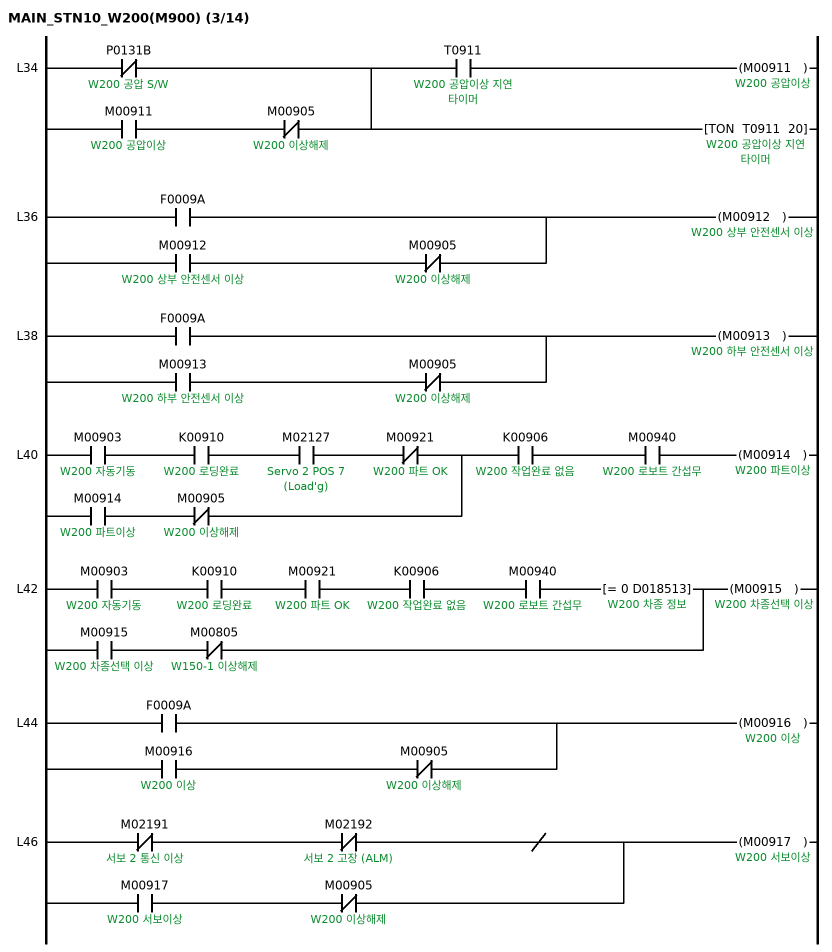
[picture p168: MAIN_STN10_W200(M900) rungs L34-L46]
; L34
LOAD NOT  P0131B	// W200 공압 S/W
LOAD      M00911	// W200 공압이상
AND NOT   M00905	// W200 이상해제
OR LOAD
MPUSH
AND       T0911	// W200 공압이상 지연 타이머
OUT       M00911	// W200 공압이상
MPOP
TON       T0911 20	// W200 공압이상 지연 타이머
; L36
LOAD      F0009A
LOAD      M00912	// W200 상부 안전센서 이상
AND NOT   M00905	// W200 이상해제
OR LOAD
OUT       M00912	// W200 상부 안전센서 이상
; L38
LOAD      F0009A
LOAD      M00913	// W200 하부 안전센서 이상
AND NOT   M00905	// W200 이상해제
OR LOAD
OUT       M00913	// W200 하부 안전센서 이상
; L40
LOAD      M00903	// W200 자동기동
AND       K00910	// W200 로딩완료
AND       M02127	// Servo 2 POS 7 (Load'g)
AND NOT   M00921	// W200 파트 OK
LOAD      M00914	// W200 파트이상
AND NOT   M00905	// W200 이상해제
OR LOAD
AND       K00906	// W200 작업완료 없음
AND       M00940	// W200 로보트 간섭무
OUT       M00914	// W200 파트이상
; L42
LOAD      M00903	// W200 자동기동
AND       K00910	// W200 로딩완료
AND       M00921	// W200 파트 OK
AND       K00906	// W200 작업완료 없음
AND       M00940	// W200 로보트 간섭무
AND=      0 D018513	// W200 차종 정보
LOAD      M00915	// W200 차종선택 이상
AND NOT   M00805	// W150-1 이상해제
OR LOAD
OUT       M00915	// W200 차종선택 이상
; L44
LOAD      F0009A
LOAD      M00916	// W200 이상
AND NOT   M00905	// W200 이상해제
OR LOAD
OUT       M00916	// W200 이상
; L46
LOAD NOT  M02191	// 서보 2 통신 이상
AND NOT   M02192	// 서보 2 고장 (ALM)
NOT
LOAD      M00917	// W200 서보이상
AND NOT   M00905	// W200 이상해제
OR LOAD
OUT       M00917	// W200 서보이상

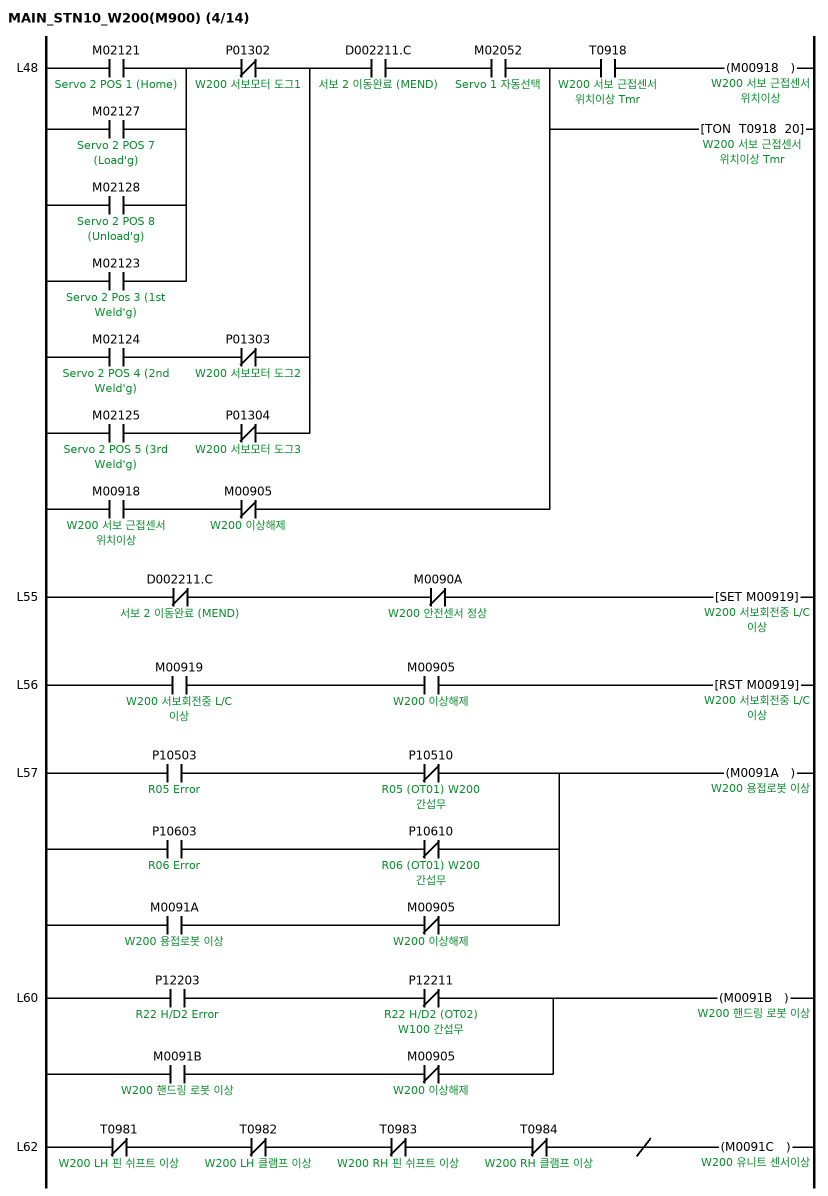
; L48
LOAD      M02121	// Servo 2 POS 1 (Home)
OR        M02127	// Servo 2 POS 7 (Load'g)
OR        M02128	// Servo 2 POS 8 (Unload'g)
OR        M02123	// Servo 2 Pos 3 (1st Weld'g)
AND NOT   P01302	// W200 서보모터 도그1
LOAD      M02124	// Servo 2 POS 4 (2nd Weld'g)
AND NOT   P01303	// W200 서보모터 도그2
OR LOAD
LOAD      M02125	// Servo 2 POS 5 (3rd Weld'g)
AND NOT   P01304	// W200 서보모터 도그3
OR LOAD
AND       D002211.C	// 서보 2 이동완료 (MEND)
AND       M02052	// Servo 1 자동선택
LOAD      M00918	// W200 서보 근접센서 위치이상
AND NOT   M00905	// W200 이상해제
OR LOAD
MPUSH
AND       T0918	// W200 서보 근접센서 위치이상 Tmr
OUT       M00918	// W200 서보 근접센서 위치이상
MPOP
TON       T0918 20	// W200 서보 근접센서 위치이상 Tmr
; L55
LOAD NOT  D002211.C	// 서보 2 이동완료 (MEND)
AND NOT   M0090A	// W200 안전센서 정상
SET       M00919	// W200 서보회전중 L/C 이상
; L56
LOAD      M00919	// W200 서보회전중 L/C 이상
AND       M00905	// W200 이상해제
RST       M00919	// W200 서보회전중 L/C 이상
; L57
LOAD      P10503	// R05 Error
AND NOT   P10510	// R05 (OT01) W200 간섭무
LOAD      P10603	// R06 Error
AND NOT   P10610	// R06 (OT01) W200 간섭무
OR LOAD
LOAD      M0091A	// W200 용접로봇 이상
AND NOT   M00905	// W200 이상해제
OR LOAD
OUT       M0091A	// W200 용접로봇 이상
; L60
LOAD      P12203	// R22 H/D2 Error
AND NOT   P12211	// R22 H/D2 (OT02) W100 간섭무
LOAD      M0091B	// W200 핸드링 로봇 이상
AND NOT   M00905	// W200 이상해제
OR LOAD
OUT       M0091B	// W200 핸드링 로봇 이상
; L62
LOAD NOT  T0981	// W200 LH 핀 쉬프트 이상
AND NOT   T0982	// W200 LH 클램프 이상
AND NOT   T0983	// W200 RH 핀 쉬프트 이상
AND NOT   T0984	// W200 RH 클램프 이상
NOT
OUT       M0091C	// W200 유니트 센서이상

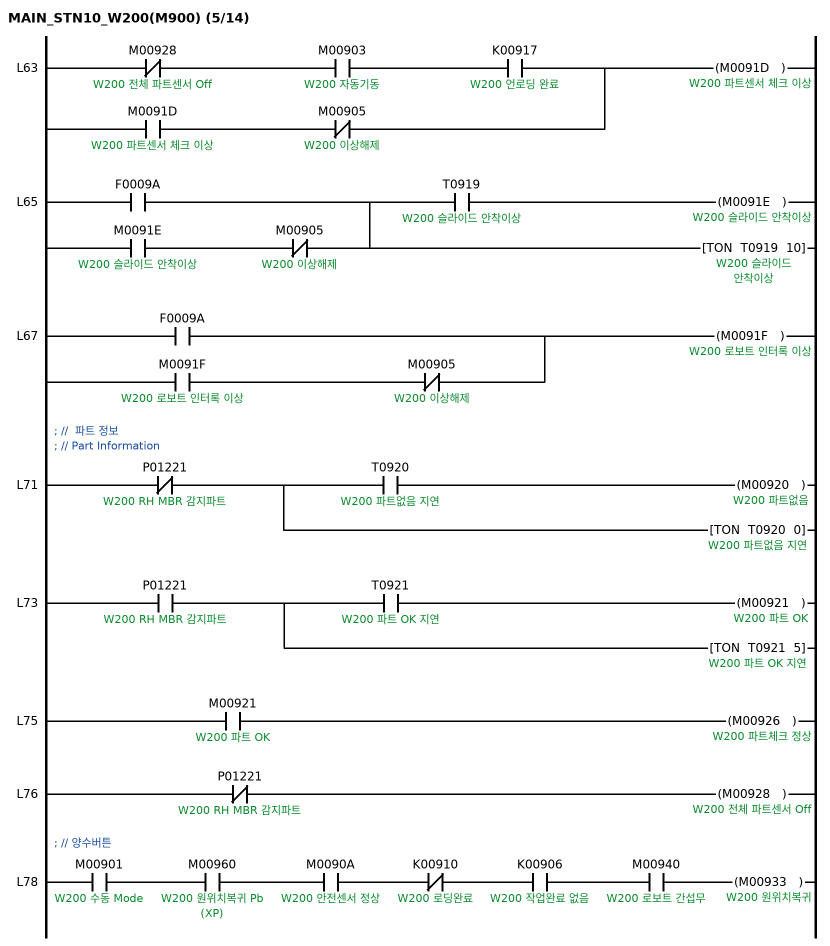
; L63
LOAD NOT  M00928	// W200 전체 파트센서 Off
AND       M00903	// W200 자동기동
AND       K00917	// W200 언로딩 완료
LOAD      M0091D	// W200 파트센서 체크 이상
AND NOT   M00905	// W200 이상해제
OR LOAD
OUT       M0091D	// W200 파트센서 체크 이상
; L65
LOAD      F0009A
LOAD      M0091E	// W200 슬라이드 안착이상
AND NOT   M00905	// W200 이상해제
OR LOAD
MPUSH
AND       T0919	// W200 슬라이드 안착이상
OUT       M0091E	// W200 슬라이드 안착이상
MPOP
TON       T0919 10	// W200 슬라이드 안착이상
; L67
LOAD      F0009A
LOAD      M0091F	// W200 로보트 인터록 이상
AND NOT   M00905	// W200 이상해제
OR LOAD
OUT       M0091F	// W200 로보트 인터록 이상
//   //  파트 정보
//   // Part Information
; L71
LOAD NOT  P01221	// W200 RH MBR 감지파트
MPUSH
AND       T0920	// W200 파트없음 지연
OUT       M00920	// W200 파트없음
MPOP
TON       T0920 0	// W200 파트없음 지연
; L73
LOAD      P01221	// W200 RH MBR 감지파트
MPUSH
AND       T0921	// W200 파트 OK 지연
OUT       M00921	// W200 파트 OK
MPOP
TON       T0921 5	// W200 파트 OK 지연
; L75
LOAD      M00921	// W200 파트 OK
OUT       M00926	// W200 파트체크 정상
; L76
LOAD NOT  P01221	// W200 RH MBR 감지파트
OUT       M00928	// W200 전체 파트센서 Off
//   // 양수버튼
; L78
LOAD      M00901	// W200 수동 Mode
AND       M00960	// W200 원위치복귀 Pb (XP)
AND       M0090A	// W200 안전센서 정상
AND NOT   K00910	// W200 로딩완료
AND       K00906	// W200 작업완료 없음
AND       M00940	// W200 로보트 간섭무
OUT       M00933	// W200 원위치복귀

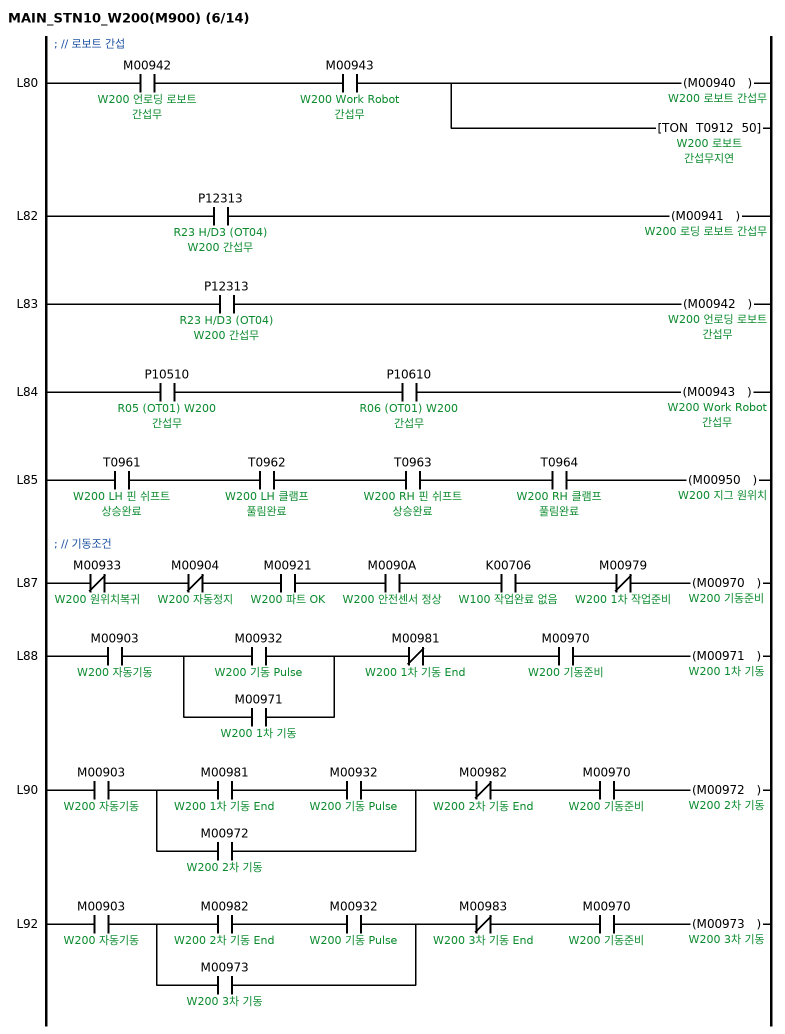
//   // 로보트 간섭
; L80
LOAD      M00942	// W200 언로딩 로보트 간섭무
AND       M00943	// W200 Work Robot 간섭무
OUT       M00940	// W200 로보트 간섭무
TON       T0912 50	// W200 로보트 간섭무지연
; L82
LOAD      P12313	// R23 H/D3 (OT04) W200 간섭무
OUT       M00941	// W200 로딩 로보트 간섭무
; L83
LOAD      P12313	// R23 H/D3 (OT04) W200 간섭무
OUT       M00942	// W200 언로딩 로보트 간섭무
; L84
LOAD      P10510	// R05 (OT01) W200 간섭무
AND       P10610	// R06 (OT01) W200 간섭무
OUT       M00943	// W200 Work Robot 간섭무
; L85
LOAD      T0961	// W200 LH 핀 쉬프트 상승완료
AND       T0962	// W200 LH 클램프 풀림완료
AND       T0963	// W200 RH 핀 쉬프트 상승완료
AND       T0964	// W200 RH 클램프 풀림완료
OUT       M00950	// W200 지그 원위치
//   // 기동조건
; L87
LOAD NOT  M00933	// W200 원위치복귀
AND NOT   M00904	// W200 자동정지
AND       M00921	// W200 파트 OK
AND       M0090A	// W200 안전센서 정상
AND       K00706	// W100 작업완료 없음
AND NOT   M00979	// W200 1차 작업준비
OUT       M00970	// W200 기동준비
; L88
LOAD      M00903	// W200 자동기동
LOAD      M00932	// W200 기동 Pulse
OR        M00971	// W200 1차 기동
AND LOAD
AND NOT   M00981	// W200 1차 기동 End
AND       M00970	// W200 기동준비
OUT       M00971	// W200 1차 기동
; L90
LOAD      M00903	// W200 자동기동
LOAD      M00981	// W200 1차 기동 End
AND       M00932	// W200 기동 Pulse
OR        M00972	// W200 2차 기동
AND LOAD
AND NOT   M00982	// W200 2차 기동 End
AND       M00970	// W200 기동준비
OUT       M00972	// W200 2차 기동
; L92
LOAD      M00903	// W200 자동기동
LOAD      M00982	// W200 2차 기동 End
AND       M00932	// W200 기동 Pulse
OR        M00973	// W200 3차 기동
AND LOAD
AND NOT   M00983	// W200 3차 기동 End
AND       M00970	// W200 기동준비
OUT       M00973	// W200 3차 기동

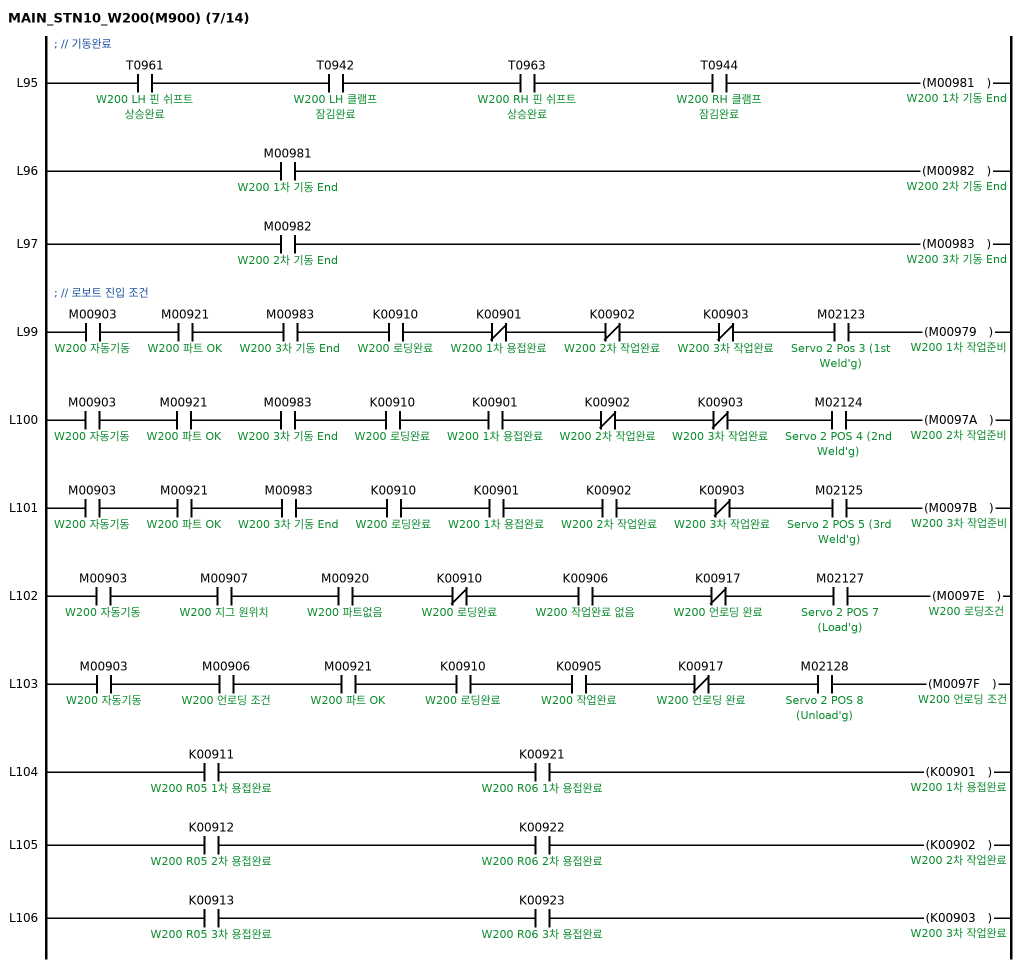
//   // 기동완료
; L95
LOAD      T0961	// W200 LH 핀 쉬프트 상승완료
AND       T0942	// W200 LH 클램프 잠김완료
AND       T0963	// W200 RH 핀 쉬프트 상승완료
AND       T0944	// W200 RH 클램프 잠김완료
OUT       M00981	// W200 1차 기동 End
; L96
LOAD      M00981	// W200 1차 기동 End
OUT       M00982	// W200 2차 기동 End
; L97
LOAD      M00982	// W200 2차 기동 End
OUT       M00983	// W200 3차 기동 End
//   // 로보트 진입 조건
; L99
LOAD      M00903	// W200 자동기동
AND       M00921	// W200 파트 OK
AND       M00983	// W200 3차 기동 End
AND       K00910	// W200 로딩완료
AND NOT   K00901	// W200 1차 용접완료
AND NOT   K00902	// W200 2차 작업완료
AND NOT   K00903	// W200 3차 작업완료
AND       M02123	// Servo 2 Pos 3 (1st Weld'g)
OUT       M00979	// W200 1차 작업준비
; L100
LOAD      M00903	// W200 자동기동
AND       M00921	// W200 파트 OK
AND       M00983	// W200 3차 기동 End
AND       K00910	// W200 로딩완료
AND       K00901	// W200 1차 용접완료
AND NOT   K00902	// W200 2차 작업완료
AND NOT   K00903	// W200 3차 작업완료
AND       M02124	// Servo 2 POS 4 (2nd Weld'g)
OUT       M0097A	// W200 2차 작업준비
; L101
LOAD      M00903	// W200 자동기동
AND       M00921	// W200 파트 OK
AND       M00983	// W200 3차 기동 End
AND       K00910	// W200 로딩완료
AND       K00901	// W200 1차 용접완료
AND       K00902	// W200 2차 작업완료
AND NOT   K00903	// W200 3차 작업완료
AND       M02125	// Servo 2 POS 5 (3rd Weld'g)
OUT       M0097B	// W200 3차 작업준비
; L102
LOAD      M00903	// W200 자동기동
AND       M00907	// W200 지그 원위치
AND       M00920	// W200 파트없음
AND NOT   K00910	// W200 로딩완료
AND       K00906	// W200 작업완료 없음
AND NOT   K00917	// W200 언로딩 완료
AND       M02127	// Servo 2 POS 7 (Load'g)
OUT       M0097E	// W200 로딩조건
; L103
LOAD      M00903	// W200 자동기동
AND       M00906	// W200 언로딩 조건
AND       M00921	// W200 파트 OK
AND       K00910	// W200 로딩완료
AND       K00905	// W200 작업완료
AND NOT   K00917	// W200 언로딩 완료
AND       M02128	// Servo 2 POS 8 (Unload'g)
OUT       M0097F	// W200 언로딩 조건
; L104
LOAD      K00911	// W200 R05 1차 용접완료
AND       K00921	// W200 R06 1차 용접완료
OUT       K00901	// W200 1차 용접완료
; L105
LOAD      K00912	// W200 R05 2차 용접완료
AND       K00922	// W200 R06 2차 용접완료
OUT       K00902	// W200 2차 작업완료
; L106
LOAD      K00913	// W200 R05 3차 용접완료
AND       K00923	// W200 R06 3차 용접완료
OUT       K00903	// W200 3차 작업완료

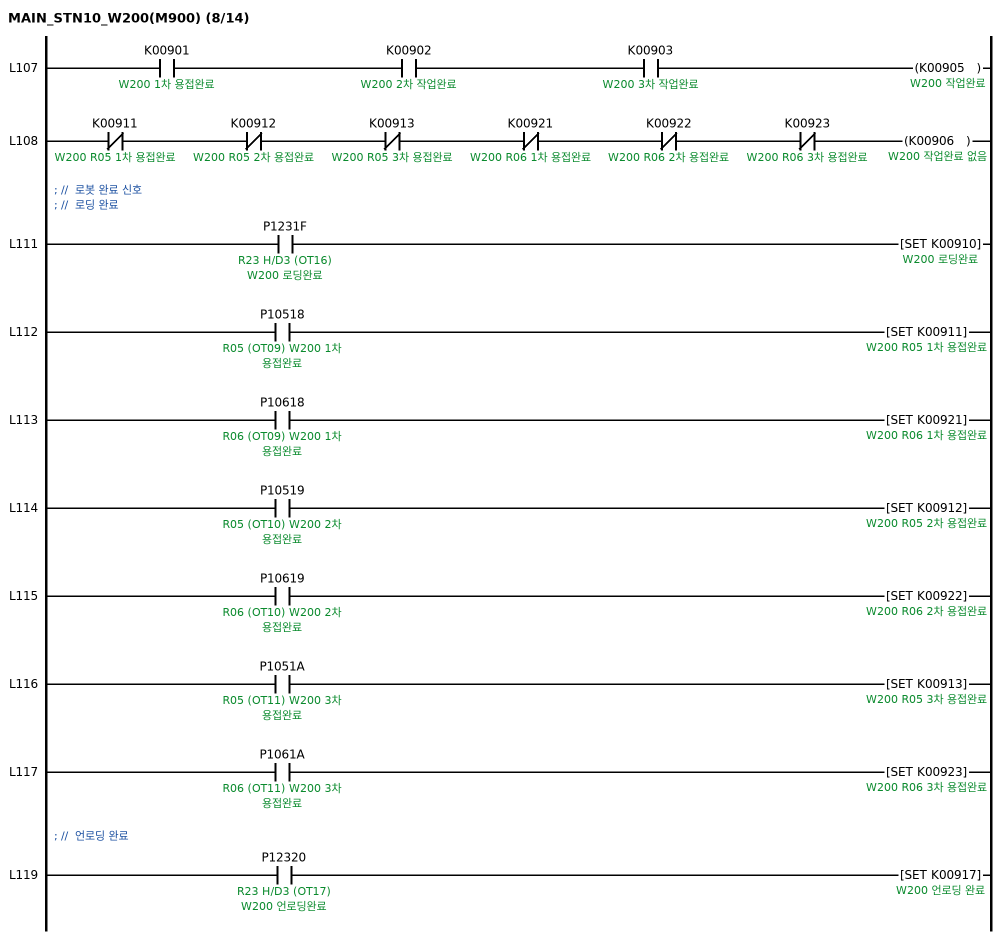
; L107
LOAD      K00901	// W200 1차 용접완료
AND       K00902	// W200 2차 작업완료
AND       K00903	// W200 3차 작업완료
OUT       K00905	// W200 작업완료
; L108
LOAD NOT  K00911	// W200 R05 1차 용접완료
AND NOT   K00912	// W200 R05 2차 용접완료
AND NOT   K00913	// W200 R05 3차 용접완료
AND NOT   K00921	// W200 R06 1차 용접완료
AND NOT   K00922	// W200 R06 2차 용접완료
AND NOT   K00923	// W200 R06 3차 용접완료
OUT       K00906	// W200 작업완료 없음
//   //  로봇 완료 신호
//   //  로딩 완료
; L111
LOAD      P1231F	// R23 H/D3 (OT16) W200 로딩완료
SET       K00910	// W200 로딩완료
; L112
LOAD      P10518	// R05 (OT09) W200 1차 용접완료
SET       K00911	// W200 R05 1차 용접완료
; L113
LOAD      P10618	// R06 (OT09) W200 1차 용접완료
SET       K00921	// W200 R06 1차 용접완료
; L114
LOAD      P10519	// R05 (OT10) W200 2차 용접완료
SET       K00912	// W200 R05 2차 용접완료
; L115
LOAD      P10619	// R06 (OT10) W200 2차 용접완료
SET       K00922	// W200 R06 2차 용접완료
; L116
LOAD      P1051A	// R05 (OT11) W200 3차 용접완료
SET       K00913	// W200 R05 3차 용접완료
; L117
LOAD      P1061A	// R06 (OT11) W200 3차 용접완료
SET       K00923	// W200 R06 3차 용접완료
//   //  언로딩 완료
; L119
LOAD      P12320	// R23 H/D3 (OT17) W200 언로딩완료
SET       K00917	// W200 언로딩 완료

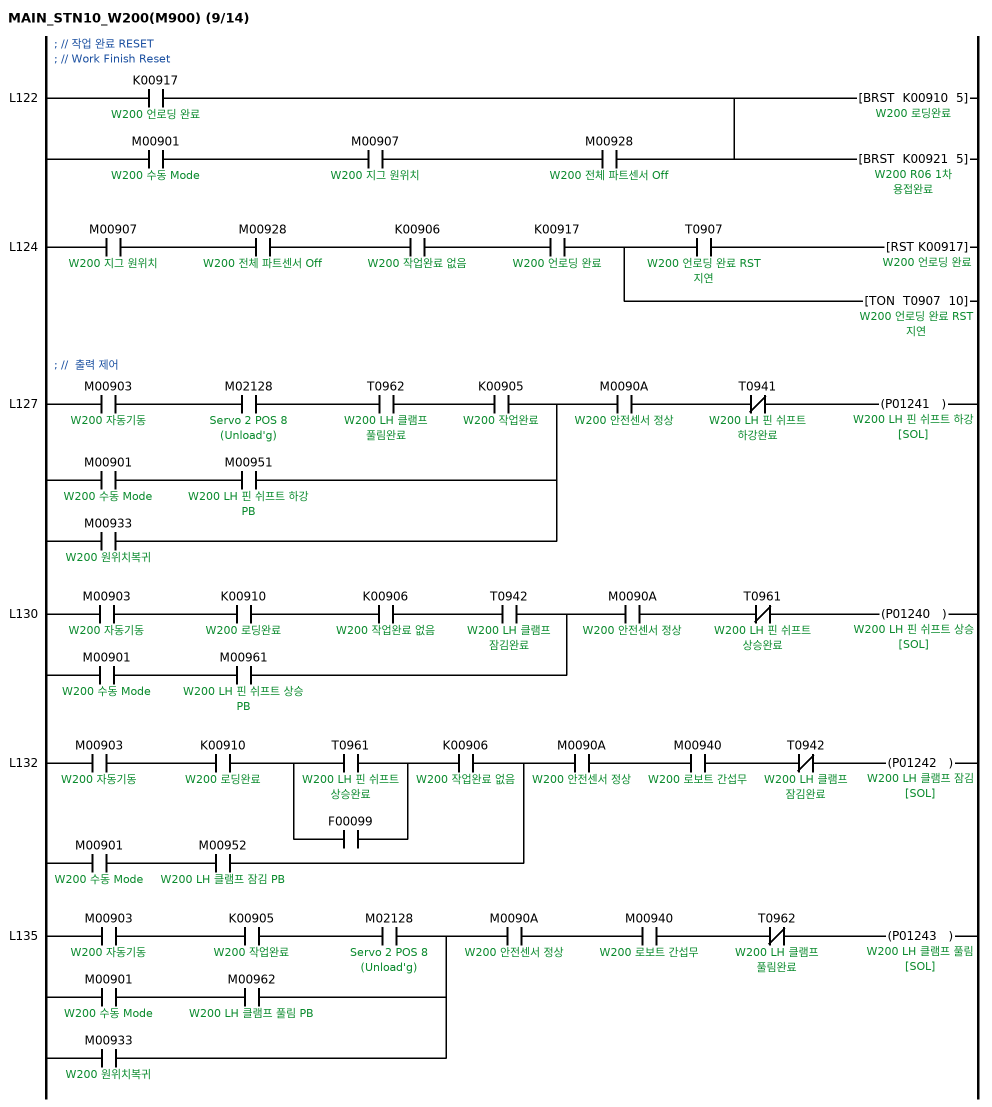
//     // 작업 완료 RESET
//   // Work Finish Reset
; L122
LOAD      K00917	// W200 언로딩 완료
LOAD      M00901	// W200 수동 Mode
AND       M00907	// W200 지그 원위치
AND       M00928	// W200 전체 파트센서 Off
OR LOAD
BRST      K00910 5	// W200 로딩완료
BRST      K00921 5	// W200 R06 1차 용접완료
; L124
LOAD      M00907	// W200 지그 원위치
AND       M00928	// W200 전체 파트센서 Off
AND       K00906	// W200 작업완료 없음
AND       K00917	// W200 언로딩 완료
MPUSH
AND       T0907	// W200 언로딩 완료 RST 지연
RST       K00917	// W200 언로딩 완료
MPOP
TON       T0907 10	// W200 언로딩 완료 RST 지연
//     //  출력 제어
; L127
LOAD      M00903	// W200 자동기동
AND       M02128	// Servo 2 POS 8 (Unload'g)
AND       T0962	// W200 LH 클램프 풀림완료
AND       K00905	// W200 작업완료
LOAD      M00901	// W200 수동 Mode
AND       M00951	// W200 LH 핀 쉬프트 하강 PB
OR LOAD
OR        M00933	// W200 원위치복귀
AND       M0090A	// W200 안전센서 정상
AND NOT   T0941	// W200 LH 핀 쉬프트 하강완료
OUT       P01241	// W200 LH 핀 쉬프트 하강 [SOL]
; L130
LOAD      M00903	// W200 자동기동
AND       K00910	// W200 로딩완료
AND       K00906	// W200 작업완료 없음
AND       T0942	// W200 LH 클램프 잠김완료
LOAD      M00901	// W200 수동 Mode
AND       M00961	// W200 LH 핀 쉬프트 상승 PB
OR LOAD
AND       M0090A	// W200 안전센서 정상
AND NOT   T0961	// W200 LH 핀 쉬프트 상승완료
OUT       P01240	// W200 LH 핀 쉬프트 상승 [SOL]
; L132
LOAD      M00903	// W200 자동기동
AND       K00910	// W200 로딩완료
LOAD      T0961	// W200 LH 핀 쉬프트 상승완료
OR        F00099
AND LOAD
AND       K00906	// W200 작업완료 없음
LOAD      M00901	// W200 수동 Mode
AND       M00952	// W200 LH 클램프 잠김 PB
OR LOAD
AND       M0090A	// W200 안전센서 정상
AND       M00940	// W200 로보트 간섭무
AND NOT   T0942	// W200 LH 클램프 잠김완료
OUT       P01242	// W200 LH 클램프 잠김 [SOL]
; L135
LOAD      M00903	// W200 자동기동
AND       K00905	// W200 작업완료
AND       M02128	// Servo 2 POS 8 (Unload'g)
LOAD      M00901	// W200 수동 Mode
AND       M00962	// W200 LH 클램프 풀림 PB
OR LOAD
OR        M00933	// W200 원위치복귀
AND       M0090A	// W200 안전센서 정상
AND       M00940	// W200 로보트 간섭무
AND NOT   T0962	// W200 LH 클램프 풀림완료
OUT       P01243	// W200 LH 클램프 풀림 [SOL]

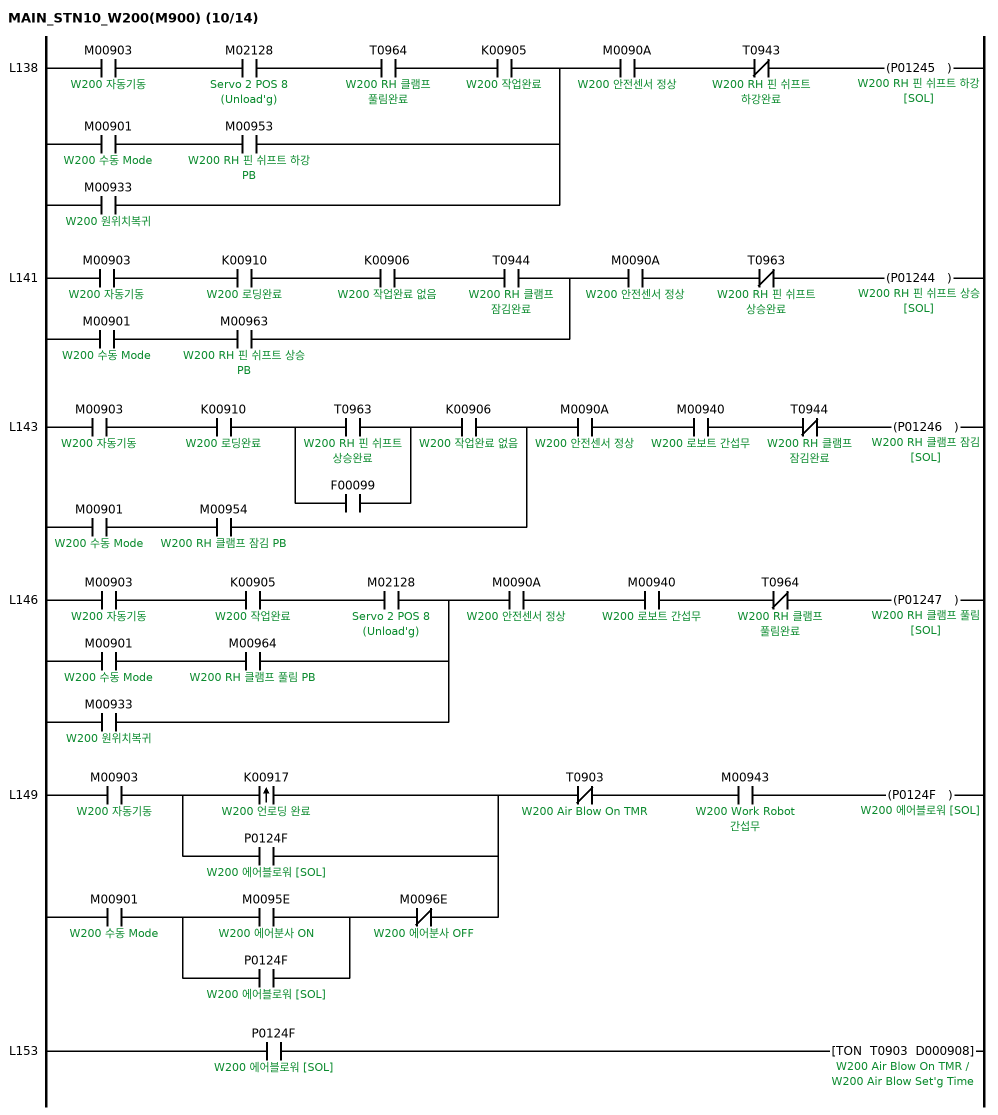
; L138
LOAD      M00903	// W200 자동기동
AND       M02128	// Servo 2 POS 8 (Unload'g)
AND       T0964	// W200 RH 클램프 풀림완료
AND       K00905	// W200 작업완료
LOAD      M00901	// W200 수동 Mode
AND       M00953	// W200 RH 핀 쉬프트 하강 PB
OR LOAD
OR        M00933	// W200 원위치복귀
AND       M0090A	// W200 안전센서 정상
AND NOT   T0943	// W200 RH 핀 쉬프트 하강완료
OUT       P01245	// W200 RH 핀 쉬프트 하강 [SOL]
; L141
LOAD      M00903	// W200 자동기동
AND       K00910	// W200 로딩완료
AND       K00906	// W200 작업완료 없음
AND       T0944	// W200 RH 클램프 잠김완료
LOAD      M00901	// W200 수동 Mode
AND       M00963	// W200 RH 핀 쉬프트 상승 PB
OR LOAD
AND       M0090A	// W200 안전센서 정상
AND NOT   T0963	// W200 RH 핀 쉬프트 상승완료
OUT       P01244	// W200 RH 핀 쉬프트 상승 [SOL]
; L143
LOAD      M00903	// W200 자동기동
AND       K00910	// W200 로딩완료
LOAD      T0963	// W200 RH 핀 쉬프트 상승완료
OR        F00099
AND LOAD
AND       K00906	// W200 작업완료 없음
LOAD      M00901	// W200 수동 Mode
AND       M00954	// W200 RH 클램프 잠김 PB
OR LOAD
AND       M0090A	// W200 안전센서 정상
AND       M00940	// W200 로보트 간섭무
AND NOT   T0944	// W200 RH 클램프 잠김완료
OUT       P01246	// W200 RH 클램프 잠김 [SOL]
; L146
LOAD      M00903	// W200 자동기동
AND       K00905	// W200 작업완료
AND       M02128	// Servo 2 POS 8 (Unload'g)
LOAD      M00901	// W200 수동 Mode
AND       M00964	// W200 RH 클램프 풀림 PB
OR LOAD
OR        M00933	// W200 원위치복귀
AND       M0090A	// W200 안전센서 정상
AND       M00940	// W200 로보트 간섭무
AND NOT   T0964	// W200 RH 클램프 풀림완료
OUT       P01247	// W200 RH 클램프 풀림 [SOL]
; L149
LOAD      M00903	// W200 자동기동
LOADP     K00917	// W200 언로딩 완료
OR        P0124F	// W200 에어블로워 [SOL]
AND LOAD
LOAD      M00901	// W200 수동 Mode
LOAD      M0095E	// W200 에어분사 ON
OR        P0124F	// W200 에어블로워 [SOL]
AND LOAD
AND NOT   M0096E	// W200 에어분사 OFF
OR LOAD
AND NOT   T0903	// W200 Air Blow On TMR
AND       M00943	// W200 Work Robot 간섭무
OUT       P0124F	// W200 에어블로워 [SOL]
; L153
LOAD      P0124F	// W200 에어블로워 [SOL]
TON       T0903 D000908	// W200 Air Blow On TMR / W200 Air Blow Set'g Time

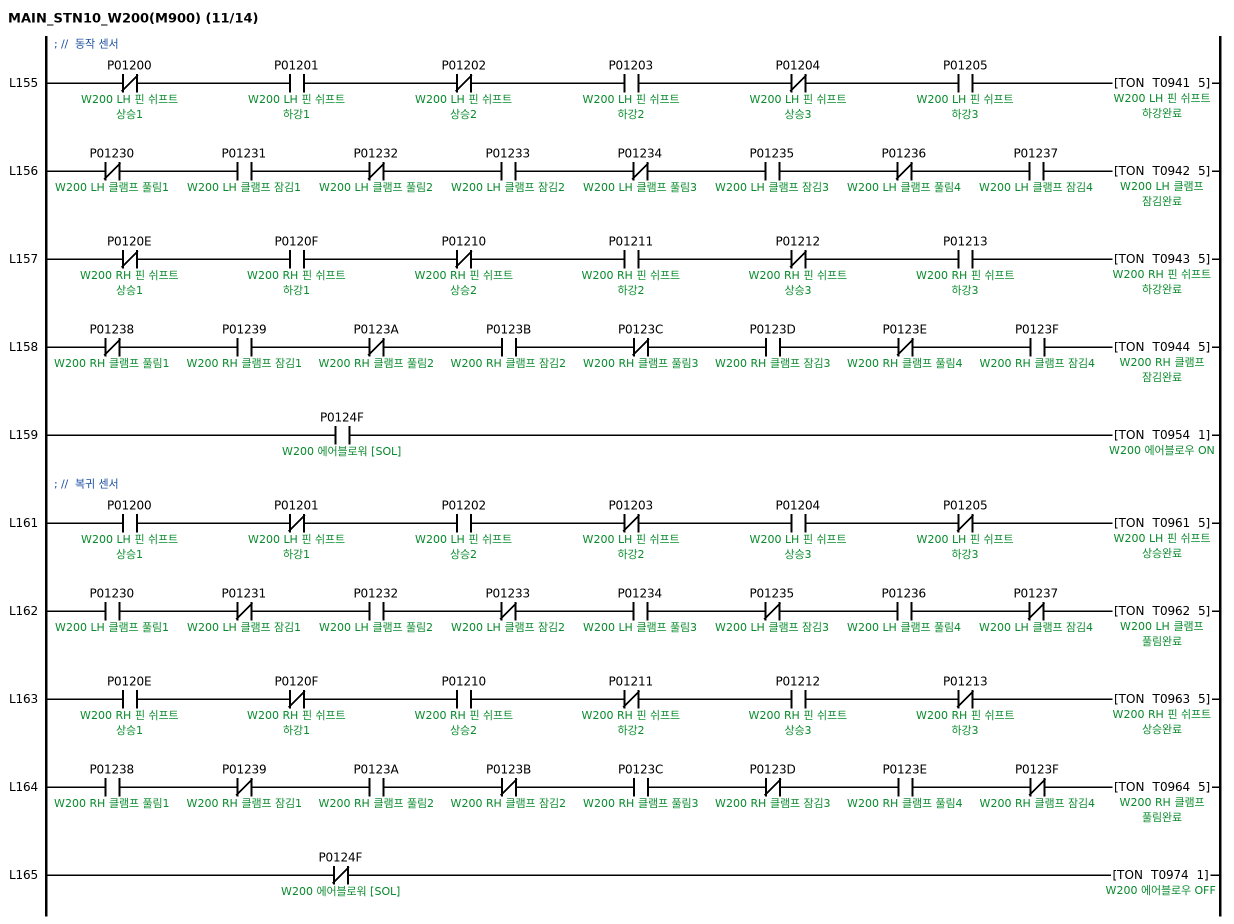
//   //  동작 센서
; L155
LOAD NOT  P01200	// W200 LH 핀 쉬프트 상승1
AND       P01201	// W200 LH 핀 쉬프트 하강1
AND NOT   P01202	// W200 LH 핀 쉬프트 상승2
AND       P01203	// W200 LH 핀 쉬프트 하강2
AND NOT   P01204	// W200 LH 핀 쉬프트 상승3
AND       P01205	// W200 LH 핀 쉬프트 하강3
TON       T0941 5	// W200 LH 핀 쉬프트 하강완료
; L156
LOAD NOT  P01230	// W200 LH 클램프 풀림1
AND       P01231	// W200 LH 클램프 잠김1
AND NOT   P01232	// W200 LH 클램프 풀림2
AND       P01233	// W200 LH 클램프 잠김2
AND NOT   P01234	// W200 LH 클램프 풀림3
AND       P01235	// W200 LH 클램프 잠김3
AND NOT   P01236	// W200 LH 클램프 풀림4
AND       P01237	// W200 LH 클램프 잠김4
TON       T0942 5	// W200 LH 클램프 잠김완료
; L157
LOAD NOT  P0120E	// W200 RH 핀 쉬프트 상승1
AND       P0120F	// W200 RH 핀 쉬프트 하강1
AND NOT   P01210	// W200 RH 핀 쉬프트 상승2
AND       P01211	// W200 RH 핀 쉬프트 하강2
AND NOT   P01212	// W200 RH 핀 쉬프트 상승3
AND       P01213	// W200 RH 핀 쉬프트 하강3
TON       T0943 5	// W200 RH 핀 쉬프트 하강완료
; L158
LOAD NOT  P01238	// W200 RH 클램프 풀림1
AND       P01239	// W200 RH 클램프 잠김1
AND NOT   P0123A	// W200 RH 클램프 풀림2
AND       P0123B	// W200 RH 클램프 잠김2
AND NOT   P0123C	// W200 RH 클램프 풀림3
AND       P0123D	// W200 RH 클램프 잠김3
AND NOT   P0123E	// W200 RH 클램프 풀림4
AND       P0123F	// W200 RH 클램프 잠김4
TON       T0944 5	// W200 RH 클램프 잠김완료
; L159
LOAD      P0124F	// W200 에어블로워 [SOL]
TON       T0954 1	// W200 에어블로우 ON
//   //  복귀 센서
; L161
LOAD      P01200	// W200 LH 핀 쉬프트 상승1
AND NOT   P01201	// W200 LH 핀 쉬프트 하강1
AND       P01202	// W200 LH 핀 쉬프트 상승2
AND NOT   P01203	// W200 LH 핀 쉬프트 하강2
AND       P01204	// W200 LH 핀 쉬프트 상승3
AND NOT   P01205	// W200 LH 핀 쉬프트 하강3
TON       T0961 5	// W200 LH 핀 쉬프트 상승완료
; L162
LOAD      P01230	// W200 LH 클램프 풀림1
AND NOT   P01231	// W200 LH 클램프 잠김1
AND       P01232	// W200 LH 클램프 풀림2
AND NOT   P01233	// W200 LH 클램프 잠김2
AND       P01234	// W200 LH 클램프 풀림3
AND NOT   P01235	// W200 LH 클램프 잠김3
AND       P01236	// W200 LH 클램프 풀림4
AND NOT   P01237	// W200 LH 클램프 잠김4
TON       T0962 5	// W200 LH 클램프 풀림완료
; L163
LOAD      P0120E	// W200 RH 핀 쉬프트 상승1
AND NOT   P0120F	// W200 RH 핀 쉬프트 하강1
AND       P01210	// W200 RH 핀 쉬프트 상승2
AND NOT   P01211	// W200 RH 핀 쉬프트 하강2
AND       P01212	// W200 RH 핀 쉬프트 상승3
AND NOT   P01213	// W200 RH 핀 쉬프트 하강3
TON       T0963 5	// W200 RH 핀 쉬프트 상승완료
; L164
LOAD      P01238	// W200 RH 클램프 풀림1
AND NOT   P01239	// W200 RH 클램프 잠김1
AND       P0123A	// W200 RH 클램프 풀림2
AND NOT   P0123B	// W200 RH 클램프 잠김2
AND       P0123C	// W200 RH 클램프 풀림3
AND NOT   P0123D	// W200 RH 클램프 잠김3
AND       P0123E	// W200 RH 클램프 풀림4
AND NOT   P0123F	// W200 RH 클램프 잠김4
TON       T0964 5	// W200 RH 클램프 풀림완료
; L165
LOAD NOT  P0124F	// W200 에어블로워 [SOL]
TON       T0974 1	// W200 에어블로우 OFF

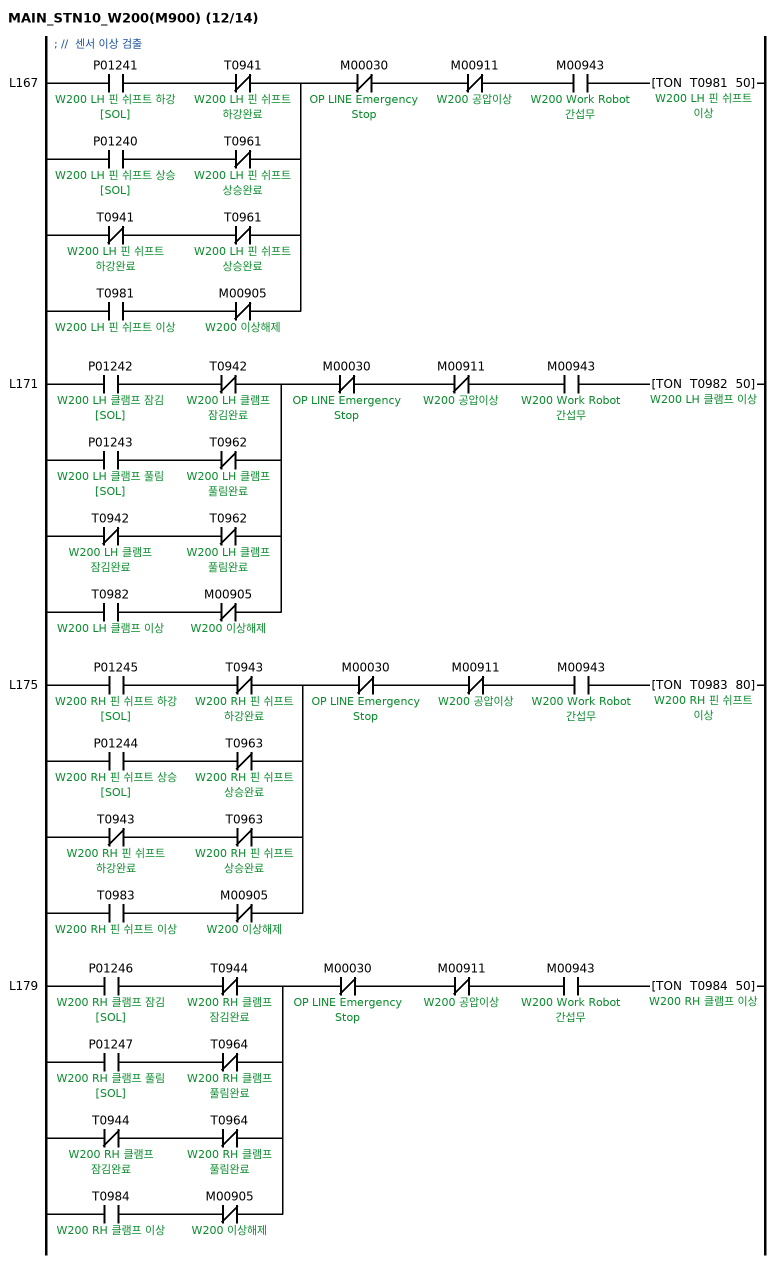
//     //  센서 이상 검출
; L167
LOAD      P01241	// W200 LH 핀 쉬프트 하강 [SOL]
AND NOT   T0941	// W200 LH 핀 쉬프트 하강완료
LOAD      P01240	// W200 LH 핀 쉬프트 상승 [SOL]
AND NOT   T0961	// W200 LH 핀 쉬프트 상승완료
OR LOAD
LOAD NOT  T0941	// W200 LH 핀 쉬프트 하강완료
AND NOT   T0961	// W200 LH 핀 쉬프트 상승완료
OR LOAD
LOAD      T0981	// W200 LH 핀 쉬프트 이상
AND NOT   M00905	// W200 이상해제
OR LOAD
AND NOT   M00030	// OP LINE Emergency Stop
AND NOT   M00911	// W200 공압이상
AND       M00943	// W200 Work Robot 간섭무
TON       T0981 50	// W200 LH 핀 쉬프트 이상
; L171
LOAD      P01242	// W200 LH 클램프 잠김 [SOL]
AND NOT   T0942	// W200 LH 클램프 잠김완료
LOAD      P01243	// W200 LH 클램프 풀림 [SOL]
AND NOT   T0962	// W200 LH 클램프 풀림완료
OR LOAD
LOAD NOT  T0942	// W200 LH 클램프 잠김완료
AND NOT   T0962	// W200 LH 클램프 풀림완료
OR LOAD
LOAD      T0982	// W200 LH 클램프 이상
AND NOT   M00905	// W200 이상해제
OR LOAD
AND NOT   M00030	// OP LINE Emergency Stop
AND NOT   M00911	// W200 공압이상
AND       M00943	// W200 Work Robot 간섭무
TON       T0982 50	// W200 LH 클램프 이상
; L175
LOAD      P01245	// W200 RH 핀 쉬프트 하강 [SOL]
AND NOT   T0943	// W200 RH 핀 쉬프트 하강완료
LOAD      P01244	// W200 RH 핀 쉬프트 상승 [SOL]
AND NOT   T0963	// W200 RH 핀 쉬프트 상승완료
OR LOAD
LOAD NOT  T0943	// W200 RH 핀 쉬프트 하강완료
AND NOT   T0963	// W200 RH 핀 쉬프트 상승완료
OR LOAD
LOAD      T0983	// W200 RH 핀 쉬프트 이상
AND NOT   M00905	// W200 이상해제
OR LOAD
AND NOT   M00030	// OP LINE Emergency Stop
AND NOT   M00911	// W200 공압이상
AND       M00943	// W200 Work Robot 간섭무
TON       T0983 80	// W200 RH 핀 쉬프트 이상
; L179
LOAD      P01246	// W200 RH 클램프 잠김 [SOL]
AND NOT   T0944	// W200 RH 클램프 잠김완료
LOAD      P01247	// W200 RH 클램프 풀림 [SOL]
AND NOT   T0964	// W200 RH 클램프 풀림완료
OR LOAD
LOAD NOT  T0944	// W200 RH 클램프 잠김완료
AND NOT   T0964	// W200 RH 클램프 풀림완료
OR LOAD
LOAD      T0984	// W200 RH 클램프 이상
AND NOT   M00905	// W200 이상해제
OR LOAD
AND NOT   M00030	// OP LINE Emergency Stop
AND NOT   M00911	// W200 공압이상
AND       M00943	// W200 Work Robot 간섭무
TON       T0984 50	// W200 RH 클램프 이상

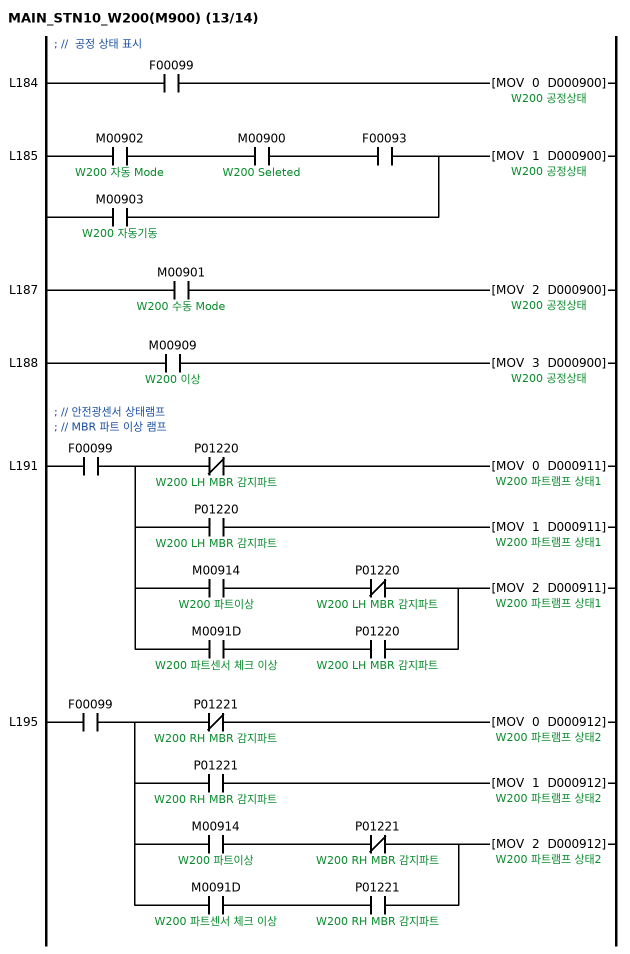
//   //  공정 상태 표시
; L184
LOAD      F00099
MOV       0 D000900	// W200 공정상태
; L185
LOAD      M00902	// W200 자동 Mode
AND       M00900	// W200 Seleted
AND       F00093
OR        M00903	// W200 자동기동
MOV       1 D000900	// W200 공정상태
; L187
LOAD      M00901	// W200 수동 Mode
MOV       2 D000900	// W200 공정상태
; L188
LOAD      M00909	// W200 이상
MOV       3 D000900	// W200 공정상태
//   // 안전광센서 상태램프
//   // MBR 파트 이상 램프
; L191
LOAD      F00099
MPUSH
AND NOT   P01220	// W200 LH MBR 감지파트
MOV       0 D000911	// W200 파트램프 상태1
MLOAD
AND       P01220	// W200 LH MBR 감지파트
MOV       1 D000911	// W200 파트램프 상태1
MPOP
LOAD      M00914	// W200 파트이상
AND NOT   P01220	// W200 LH MBR 감지파트
LOAD      M0091D	// W200 파트센서 체크 이상
AND       P01220	// W200 LH MBR 감지파트
OR LOAD
AND LOAD
MOV       2 D000911	// W200 파트램프 상태1
; L195
LOAD      F00099
MPUSH
AND NOT   P01221	// W200 RH MBR 감지파트
MOV       0 D000912	// W200 파트램프 상태2
MLOAD
AND       P01221	// W200 RH MBR 감지파트
MOV       1 D000912	// W200 파트램프 상태2
MPOP
LOAD      M00914	// W200 파트이상
AND NOT   P01221	// W200 RH MBR 감지파트
LOAD      M0091D	// W200 파트센서 체크 이상
AND       P01221	// W200 RH MBR 감지파트
OR LOAD
AND LOAD
MOV       2 D000912	// W200 파트램프 상태2

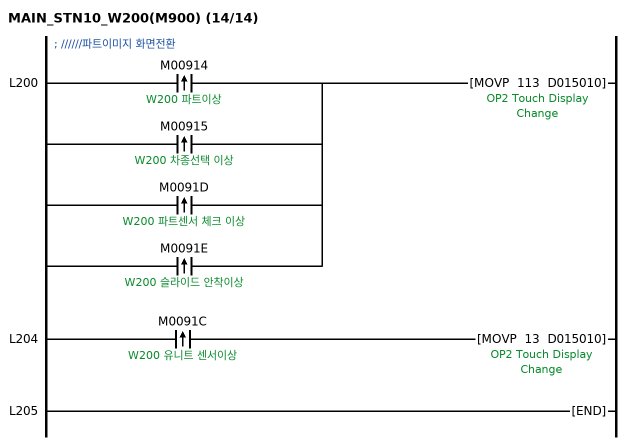
// //////파트이미지 화면전환
; L200
LOADP     M00914	// W200 파트이상
ORP       M00915	// W200 차종선택 이상
ORP       M0091D	// W200 파트센서 체크 이상
ORP       M0091E	// W200 슬라이드 안착이상
MOVP      113 D015010	// OP2 Touch Display Change
; L204
LOADP     M0091C	// W200 유니트 센서이상
MOVP      13 D015010	// OP2 Touch Display Change
; L205
END

PROGRAM MAIN_STN11_W250(M1000) (task: 스캔 프로그램)

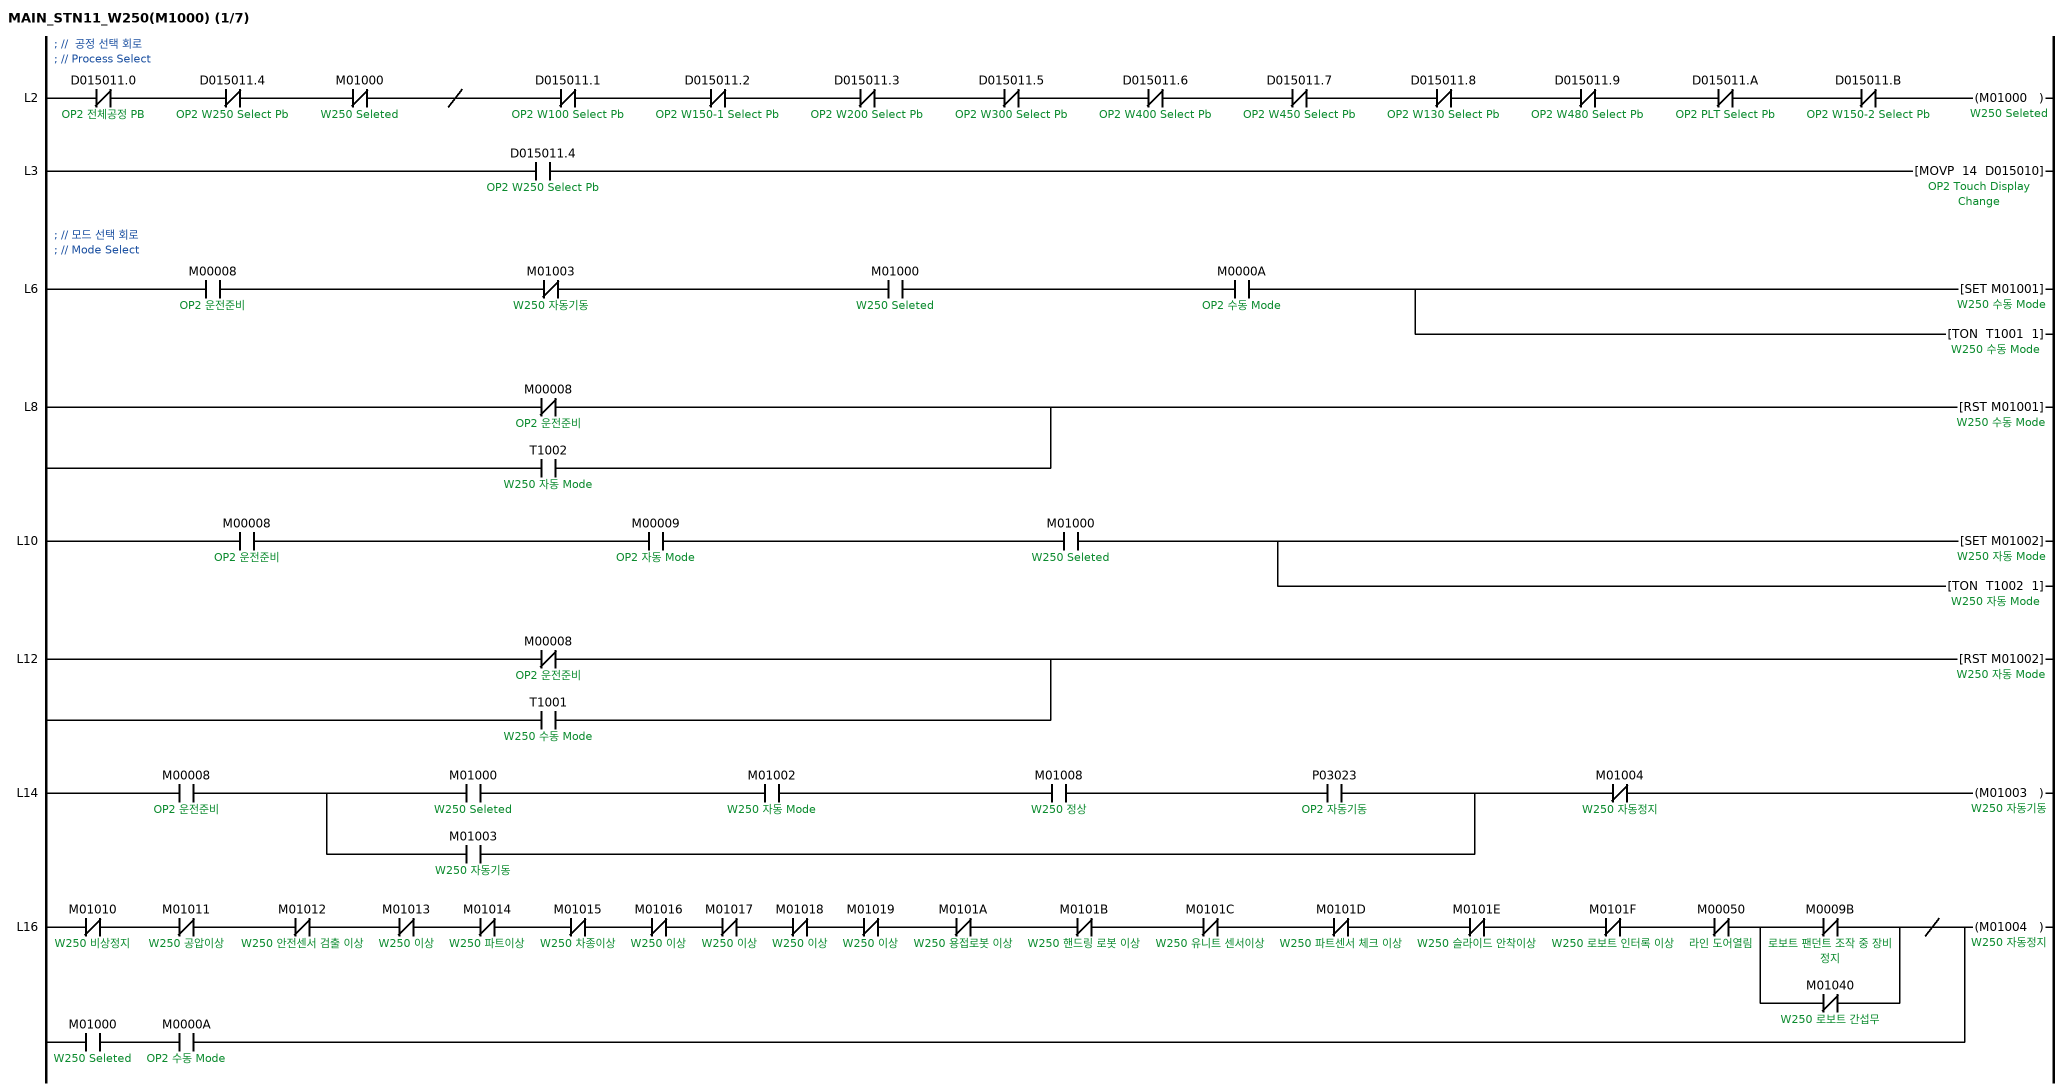
//   //  공정 선택 회로
//   // Process Select
; L2
LOAD NOT  D015011.0	// OP2 전체공정 PB
AND NOT   D015011.4	// OP2 W250 Select Pb
AND NOT   M01000	// W250 Seleted
NOT
AND NOT   D015011.1	// OP2 W100 Select Pb
AND NOT   D015011.2	// OP2 W150-1 Select Pb
AND NOT   D015011.3	// OP2 W200 Select Pb
AND NOT   D015011.5	// OP2 W300 Select Pb
AND NOT   D015011.6	// OP2 W400 Select Pb
AND NOT   D015011.7	// OP2 W450 Select Pb
AND NOT   D015011.8	// OP2 W130 Select Pb
AND NOT   D015011.9	// OP2 W480 Select Pb
AND NOT   D015011.A	// OP2 PLT Select Pb
AND NOT   D015011.B	// OP2 W150-2 Select Pb
OUT       M01000	// W250 Seleted
; L3
LOAD      D015011.4	// OP2 W250 Select Pb
MOVP      14 D015010	// OP2 Touch Display Change
// // 모드 선택 회로
//   // Mode Select
; L6
LOAD      M00008	// OP2 운전준비
AND NOT   M01003	// W250 자동기동
AND       M01000	// W250 Seleted
AND       M0000A	// OP2 수동 Mode
SET       M01001	// W250 수동 Mode
TON       T1001 1	// W250 수동 Mode
; L8
LOAD NOT  M00008	// OP2 운전준비
OR        T1002	// W250 자동 Mode
RST       M01001	// W250 수동 Mode
; L10
LOAD      M00008	// OP2 운전준비
AND       M00009	// OP2 자동 Mode
AND       M01000	// W250 Seleted
SET       M01002	// W250 자동 Mode
TON       T1002 1	// W250 자동 Mode
; L12
LOAD NOT  M00008	// OP2 운전준비
OR        T1001	// W250 수동 Mode
RST       M01002	// W250 자동 Mode
; L14
LOAD      M00008	// OP2 운전준비
LOAD      M01000	// W250 Seleted
AND       M01002	// W250 자동 Mode
AND       M01008	// W250 정상
AND       P03023	// OP2 자동기동
OR        M01003	// W250 자동기동
AND LOAD
AND NOT   M01004	// W250 자동정지
OUT       M01003	// W250 자동기동
; L16
LOAD NOT  M01010	// W250 비상정지
AND NOT   M01011	// W250 공압이상
AND NOT   M01012	// W250 안전센서 검출 이상
AND NOT   M01013	// W250 이상
AND NOT   M01014	// W250 파트이상
AND NOT   M01015	// W250 차종이상
AND NOT   M01016	// W250 이상
AND NOT   M01017	// W250 이상
AND NOT   M01018	// W250 이상
AND NOT   M01019	// W250 이상
AND NOT   M0101A	// W250 용접로봇 이상
AND NOT   M0101B	// W250 핸드링 로봇 이상
AND NOT   M0101C	// W250 유니트 센서이상
AND NOT   M0101D	// W250 파트센서 체크 이상
AND NOT   M0101E	// W250 슬라이드 안착이상
AND NOT   M0101F	// W250 로보트 인터록 이상
AND NOT   M00050	// 라인 도어열림
LOAD NOT  M0009B	// 로보트 팬던트 조작 중 장비 정지
OR NOT    M01040	// W250 로보트 간섭무
AND LOAD
NOT
LOAD      M01000	// W250 Seleted
AND       M0000A	// OP2 수동 Mode
OR LOAD
OUT       M01004	// W250 자동정지

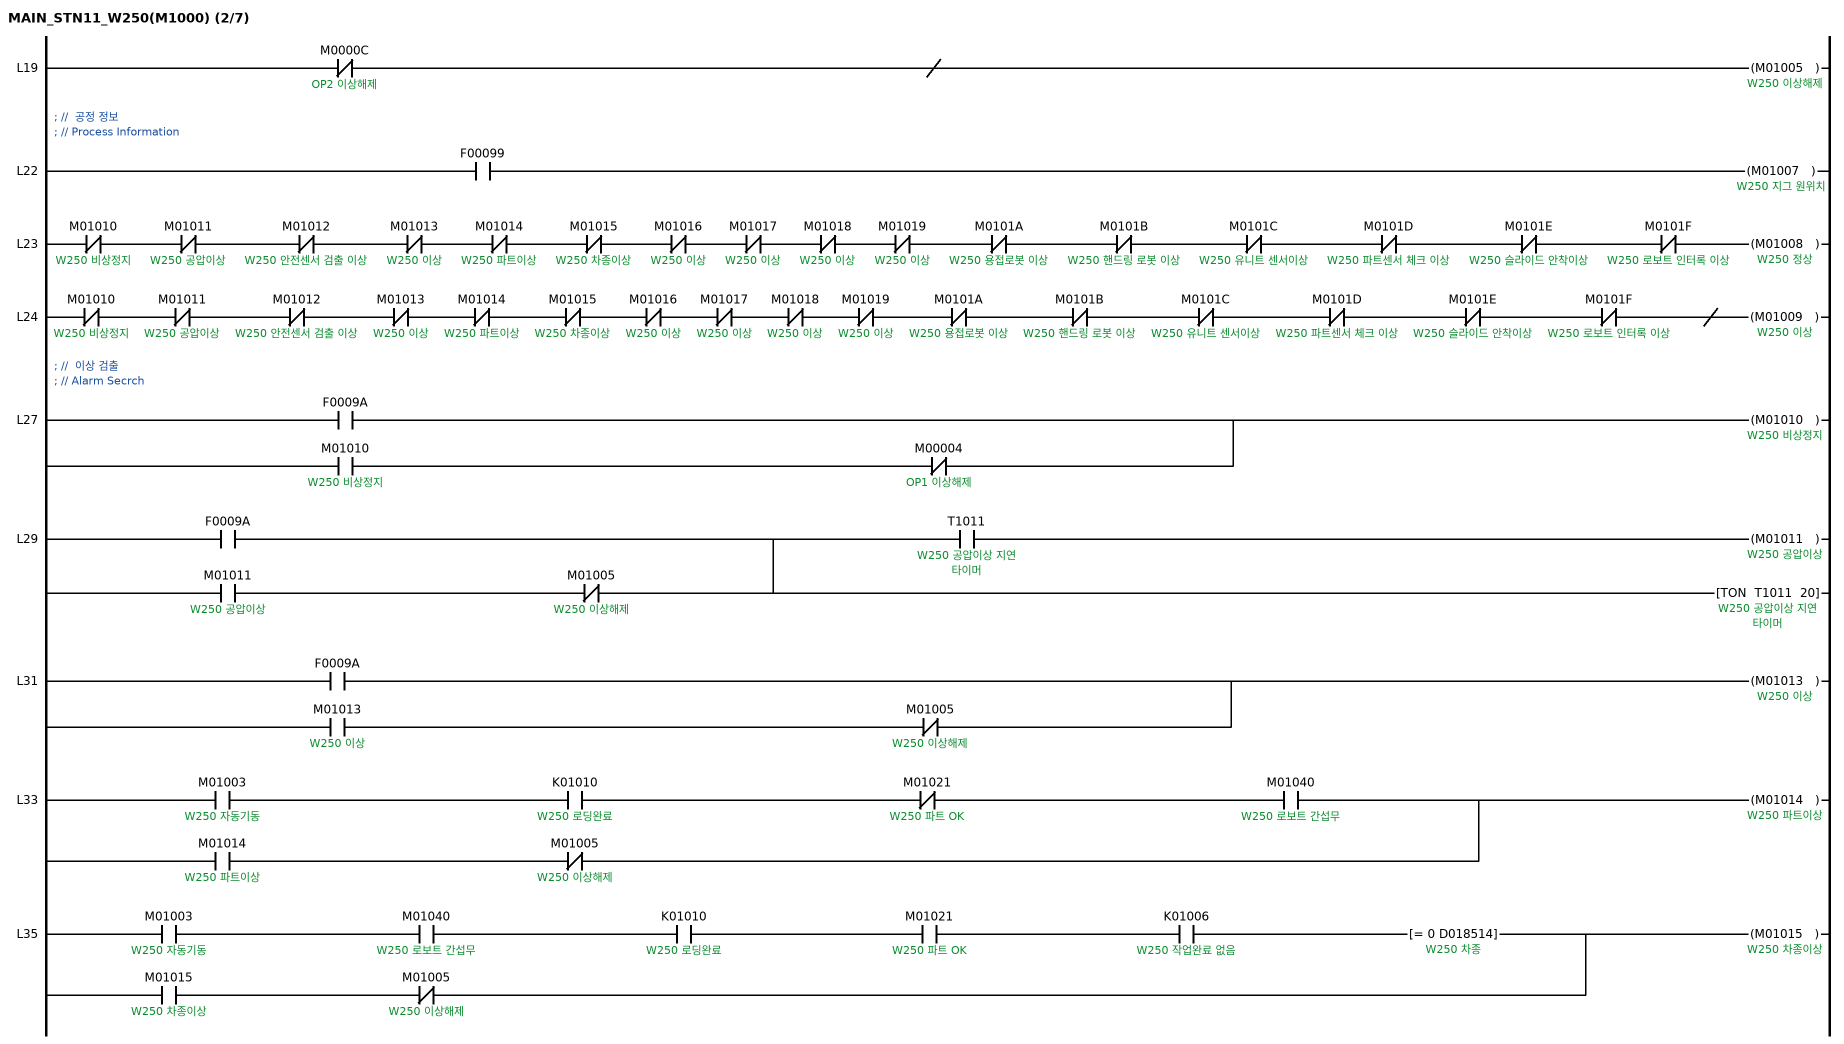
; L19
LOAD NOT  M0000C	// OP2 이상해제
NOT
OUT       M01005	// W250 이상해제
//   //  공정 정보
//   // Process Information
; L22
LOAD      F00099
OUT       M01007	// W250 지그 원위치
; L23
LOAD NOT  M01010	// W250 비상정지
AND NOT   M01011	// W250 공압이상
AND NOT   M01012	// W250 안전센서 검출 이상
AND NOT   M01013	// W250 이상
AND NOT   M01014	// W250 파트이상
AND NOT   M01015	// W250 차종이상
AND NOT   M01016	// W250 이상
AND NOT   M01017	// W250 이상
AND NOT   M01018	// W250 이상
AND NOT   M01019	// W250 이상
AND NOT   M0101A	// W250 용접로봇 이상
AND NOT   M0101B	// W250 핸드링 로봇 이상
AND NOT   M0101C	// W250 유니트 센서이상
AND NOT   M0101D	// W250 파트센서 체크 이상
AND NOT   M0101E	// W250 슬라이드 안착이상
AND NOT   M0101F	// W250 로보트 인터록 이상
OUT       M01008	// W250 정상
; L24
LOAD NOT  M01010	// W250 비상정지
AND NOT   M01011	// W250 공압이상
AND NOT   M01012	// W250 안전센서 검출 이상
AND NOT   M01013	// W250 이상
AND NOT   M01014	// W250 파트이상
AND NOT   M01015	// W250 차종이상
AND NOT   M01016	// W250 이상
AND NOT   M01017	// W250 이상
AND NOT   M01018	// W250 이상
AND NOT   M01019	// W250 이상
AND NOT   M0101A	// W250 용접로봇 이상
AND NOT   M0101B	// W250 핸드링 로봇 이상
AND NOT   M0101C	// W250 유니트 센서이상
AND NOT   M0101D	// W250 파트센서 체크 이상
AND NOT   M0101E	// W250 슬라이드 안착이상
AND NOT   M0101F	// W250 로보트 인터록 이상
NOT
OUT       M01009	// W250 이상
//   //  이상 검출
//   // Alarm Secrch
; L27
LOAD      F0009A
LOAD      M01010	// W250 비상정지
AND NOT   M00004	// OP1 이상해제
OR LOAD
OUT       M01010	// W250 비상정지
; L29
LOAD      F0009A
LOAD      M01011	// W250 공압이상
AND NOT   M01005	// W250 이상해제
OR LOAD
MPUSH
AND       T1011	// W250 공압이상 지연 타이머
OUT       M01011	// W250 공압이상
MPOP
TON       T1011 20	// W250 공압이상 지연 타이머
; L31
LOAD      F0009A
LOAD      M01013	// W250 이상
AND NOT   M01005	// W250 이상해제
OR LOAD
OUT       M01013	// W250 이상
; L33
LOAD      M01003	// W250 자동기동
AND       K01010	// W250 로딩완료
AND NOT   M01021	// W250 파트 OK
AND       M01040	// W250 로보트 간섭무
LOAD      M01014	// W250 파트이상
AND NOT   M01005	// W250 이상해제
OR LOAD
OUT       M01014	// W250 파트이상
; L35
LOAD      M01003	// W250 자동기동
AND       M01040	// W250 로보트 간섭무
AND       K01010	// W250 로딩완료
AND       M01021	// W250 파트 OK
AND       K01006	// W250 작업완료 없음
AND=      0 D018514	// W250 차종
LOAD      M01015	// W250 차종이상
AND NOT   M01005	// W250 이상해제
OR LOAD
OUT       M01015	// W250 차종이상

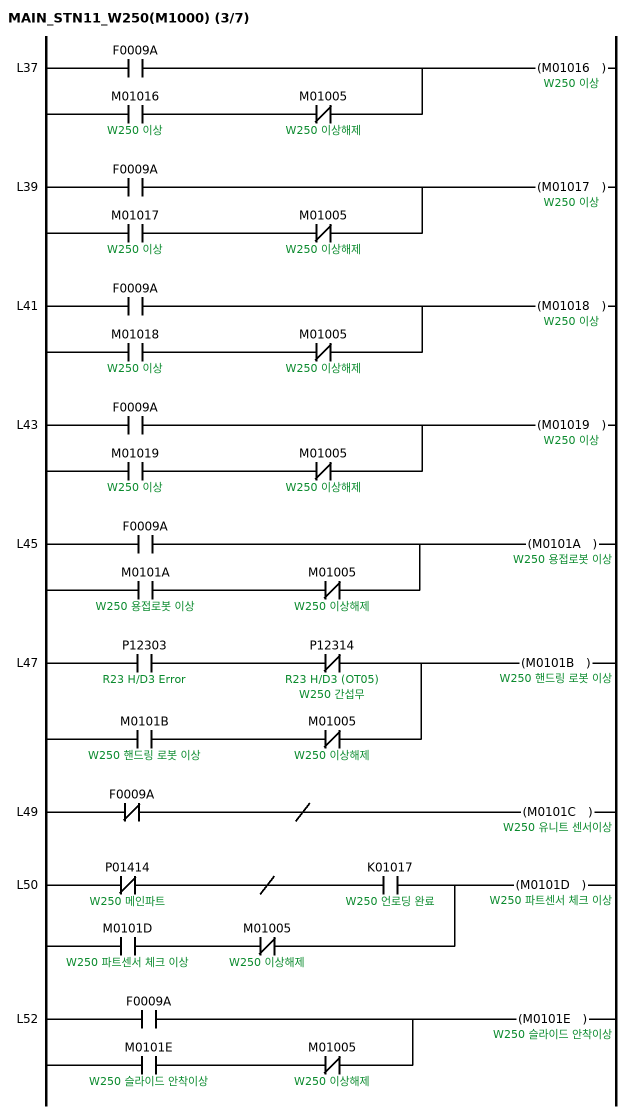
; L37
LOAD      F0009A
LOAD      M01016	// W250 이상
AND NOT   M01005	// W250 이상해제
OR LOAD
OUT       M01016	// W250 이상
; L39
LOAD      F0009A
LOAD      M01017	// W250 이상
AND NOT   M01005	// W250 이상해제
OR LOAD
OUT       M01017	// W250 이상
; L41
LOAD      F0009A
LOAD      M01018	// W250 이상
AND NOT   M01005	// W250 이상해제
OR LOAD
OUT       M01018	// W250 이상
; L43
LOAD      F0009A
LOAD      M01019	// W250 이상
AND NOT   M01005	// W250 이상해제
OR LOAD
OUT       M01019	// W250 이상
; L45
LOAD      F0009A
LOAD      M0101A	// W250 용접로봇 이상
AND NOT   M01005	// W250 이상해제
OR LOAD
OUT       M0101A	// W250 용접로봇 이상
; L47
LOAD      P12303	// R23 H/D3 Error
AND NOT   P12314	// R23 H/D3 (OT05) W250 간섭무
LOAD      M0101B	// W250 핸드링 로봇 이상
AND NOT   M01005	// W250 이상해제
OR LOAD
OUT       M0101B	// W250 핸드링 로봇 이상
; L49
LOAD NOT  F0009A
NOT
OUT       M0101C	// W250 유니트 센서이상
; L50
LOAD NOT  P01414	// W250 메인파트
NOT
AND       K01017	// W250 언로딩 완료
LOAD      M0101D	// W250 파트센서 체크 이상
AND NOT   M01005	// W250 이상해제
OR LOAD
OUT       M0101D	// W250 파트센서 체크 이상
; L52
LOAD      F0009A
LOAD      M0101E	// W250 슬라이드 안착이상
AND NOT   M01005	// W250 이상해제
OR LOAD
OUT       M0101E	// W250 슬라이드 안착이상

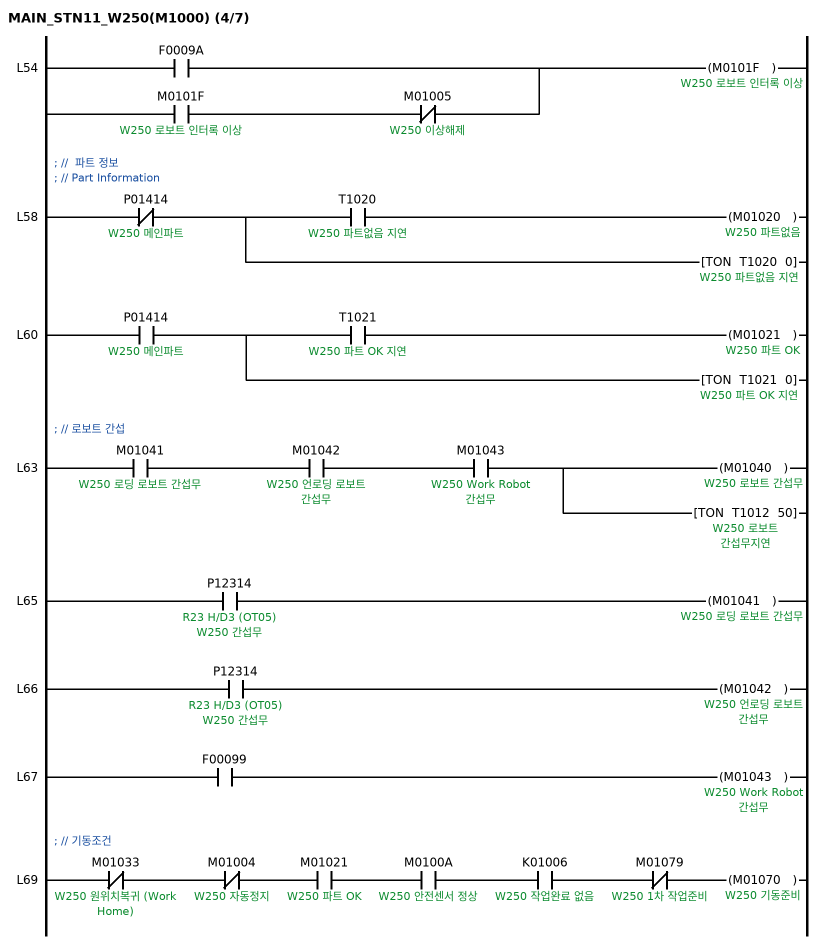
; L54
LOAD      F0009A
LOAD      M0101F	// W250 로보트 인터록 이상
AND NOT   M01005	// W250 이상해제
OR LOAD
OUT       M0101F	// W250 로보트 인터록 이상
//   //  파트 정보
//   // Part Information
; L58
LOAD NOT  P01414	// W250 메인파트
MPUSH
AND       T1020	// W250 파트없음 지연
OUT       M01020	// W250 파트없음
MPOP
TON       T1020 0	// W250 파트없음 지연
; L60
LOAD      P01414	// W250 메인파트
MPUSH
AND       T1021	// W250 파트 OK 지연
OUT       M01021	// W250 파트 OK
MPOP
TON       T1021 0	// W250 파트 OK 지연
//   // 로보트 간섭
; L63
LOAD      M01041	// W250 로딩 로보트 간섭무
AND       M01042	// W250 언로딩 로보트 간섭무
AND       M01043	// W250 Work Robot 간섭무
OUT       M01040	// W250 로보트 간섭무
TON       T1012 50	// W250 로보트 간섭무지연
; L65
LOAD      P12314	// R23 H/D3 (OT05) W250 간섭무
OUT       M01041	// W250 로딩 로보트 간섭무
; L66
LOAD      P12314	// R23 H/D3 (OT05) W250 간섭무
OUT       M01042	// W250 언로딩 로보트 간섭무
; L67
LOAD      F00099
OUT       M01043	// W250 Work Robot 간섭무
//   // 기동조건
; L69
LOAD NOT  M01033	// W250 원위치복귀 (Work Home)
AND NOT   M01004	// W250 자동정지
AND       M01021	// W250 파트 OK
AND       M0100A	// W250 안전센서 정상
AND       K01006	// W250 작업완료 없음
AND NOT   M01079	// W250 1차 작업준비
OUT       M01070	// W250 기동준비

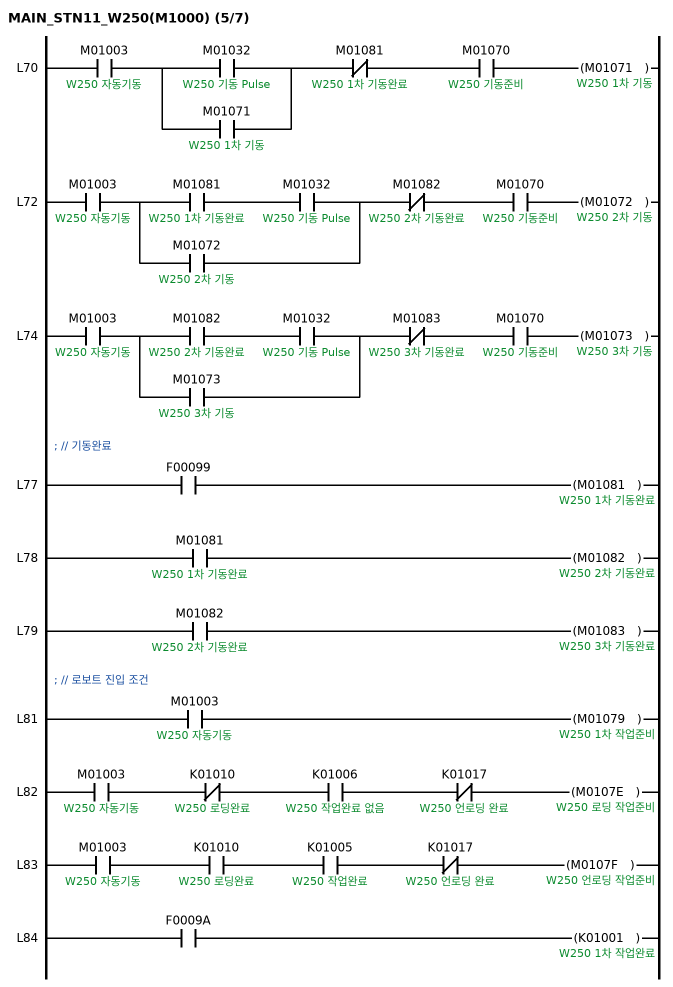
; L70
LOAD      M01003	// W250 자동기동
LOAD      M01032	// W250 기동 Pulse
OR        M01071	// W250 1차 기동
AND LOAD
AND NOT   M01081	// W250 1차 기동완료
AND       M01070	// W250 기동준비
OUT       M01071	// W250 1차 기동
; L72
LOAD      M01003	// W250 자동기동
LOAD      M01081	// W250 1차 기동완료
AND       M01032	// W250 기동 Pulse
OR        M01072	// W250 2차 기동
AND LOAD
AND NOT   M01082	// W250 2차 기동완료
AND       M01070	// W250 기동준비
OUT       M01072	// W250 2차 기동
; L74
LOAD      M01003	// W250 자동기동
LOAD      M01082	// W250 2차 기동완료
AND       M01032	// W250 기동 Pulse
OR        M01073	// W250 3차 기동
AND LOAD
AND NOT   M01083	// W250 3차 기동완료
AND       M01070	// W250 기동준비
OUT       M01073	// W250 3차 기동
//   // 기동완료
; L77
LOAD      F00099
OUT       M01081	// W250 1차 기동완료
; L78
LOAD      M01081	// W250 1차 기동완료
OUT       M01082	// W250 2차 기동완료
; L79
LOAD      M01082	// W250 2차 기동완료
OUT       M01083	// W250 3차 기동완료
//   // 로보트 진입 조건
; L81
LOAD      M01003	// W250 자동기동
OUT       M01079	// W250 1차 작업준비
; L82
LOAD      M01003	// W250 자동기동
AND NOT   K01010	// W250 로딩완료
AND       K01006	// W250 작업완료 없음
AND NOT   K01017	// W250 언로딩 완료
OUT       M0107E	// W250 로딩 작업준비
; L83
LOAD      M01003	// W250 자동기동
AND       K01010	// W250 로딩완료
AND       K01005	// W250 작업완료
AND NOT   K01017	// W250 언로딩 완료
OUT       M0107F	// W250 언로딩 작업준비
; L84
LOAD      F0009A
OUT       K01001	// W250 1차 작업완료

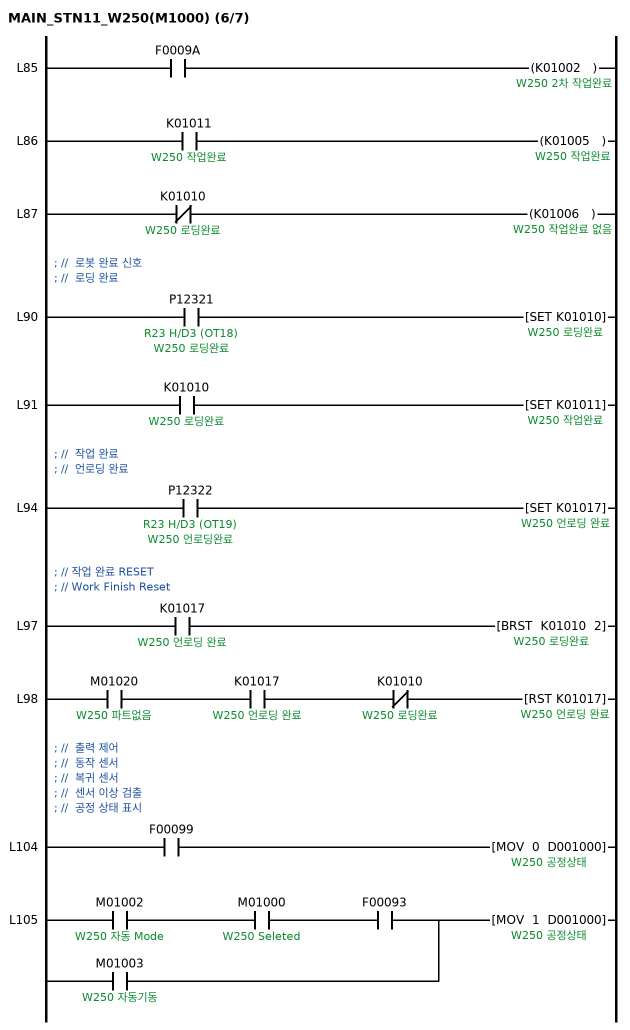
; L85
LOAD      F0009A
OUT       K01002	// W250 2차 작업완료
; L86
LOAD      K01011	// W250 작업완료
OUT       K01005	// W250 작업완료
; L87
LOAD NOT  K01010	// W250 로딩완료
OUT       K01006	// W250 작업완료 없음
//   //  로봇 완료 신호
//   //  로딩 완료
; L90
LOAD      P12321	// R23 H/D3 (OT18) W250 로딩완료
SET       K01010	// W250 로딩완료
; L91
LOAD      K01010	// W250 로딩완료
SET       K01011	// W250 작업완료
//   //  작업 완료
//   //  언로딩 완료
; L94
LOAD      P12322	// R23 H/D3 (OT19) W250 언로딩완료
SET       K01017	// W250 언로딩 완료
//     // 작업 완료 RESET
//   // Work Finish Reset
; L97
LOAD      K01017	// W250 언로딩 완료
BRST      K01010 2	// W250 로딩완료
; L98
LOAD      M01020	// W250 파트없음
AND       K01017	// W250 언로딩 완료
AND NOT   K01010	// W250 로딩완료
RST       K01017	// W250 언로딩 완료
//     //  출력 제어
//   //  동작 센서
//   //  복귀 센서
//     //  센서 이상 검출
//   //  공정 상태 표시
; L104
LOAD      F00099
MOV       0 D001000	// W250 공정상태
; L105
LOAD      M01002	// W250 자동 Mode
AND       M01000	// W250 Seleted
AND       F00093
OR        M01003	// W250 자동기동
MOV       1 D001000	// W250 공정상태

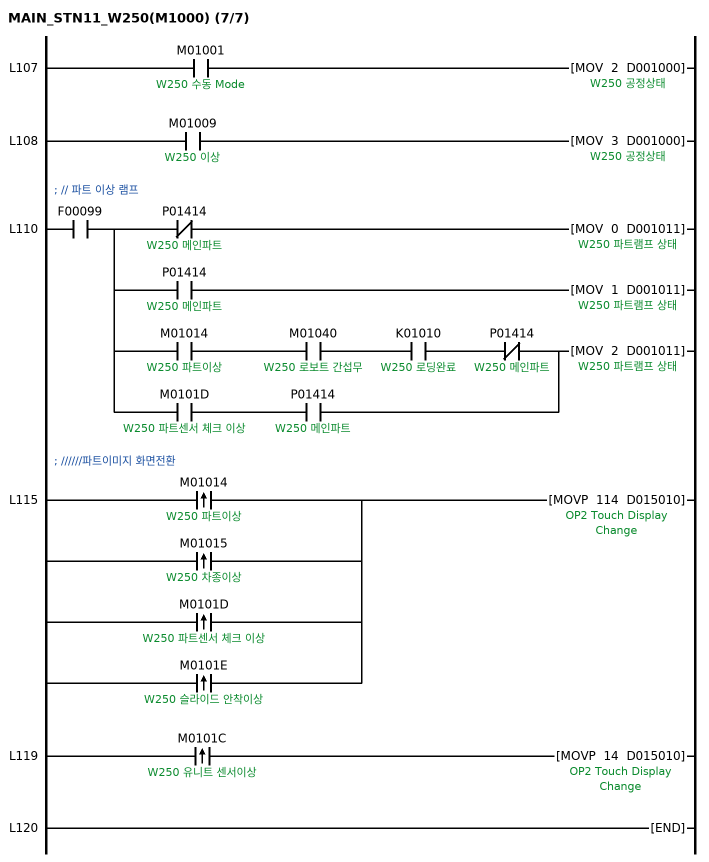
; L107
LOAD      M01001	// W250 수동 Mode
MOV       2 D001000	// W250 공정상태
; L108
LOAD      M01009	// W250 이상
MOV       3 D001000	// W250 공정상태
//   // 파트 이상 램프
; L110
LOAD      F00099
MPUSH
AND NOT   P01414	// W250 메인파트
MOV       0 D001011	// W250 파트램프 상태
MLOAD
AND       P01414	// W250 메인파트
MOV       1 D001011	// W250 파트램프 상태
MPOP
LOAD      M01014	// W250 파트이상
AND       M01040	// W250 로보트 간섭무
AND       K01010	// W250 로딩완료
AND NOT   P01414	// W250 메인파트
LOAD      M0101D	// W250 파트센서 체크 이상
AND       P01414	// W250 메인파트
OR LOAD
AND LOAD
MOV       2 D001011	// W250 파트램프 상태
// //////파트이미지 화면전환
; L115
LOADP     M01014	// W250 파트이상
ORP       M01015	// W250 차종이상
ORP       M0101D	// W250 파트센서 체크 이상
ORP       M0101E	// W250 슬라이드 안착이상
MOVP      114 D015010	// OP2 Touch Display Change
; L119
LOADP     M0101C	// W250 유니트 센서이상
MOVP      14 D015010	// OP2 Touch Display Change
; L120
END

PROGRAM MAIN_STN12_W300(M1100) (task: 스캔 프로그램)

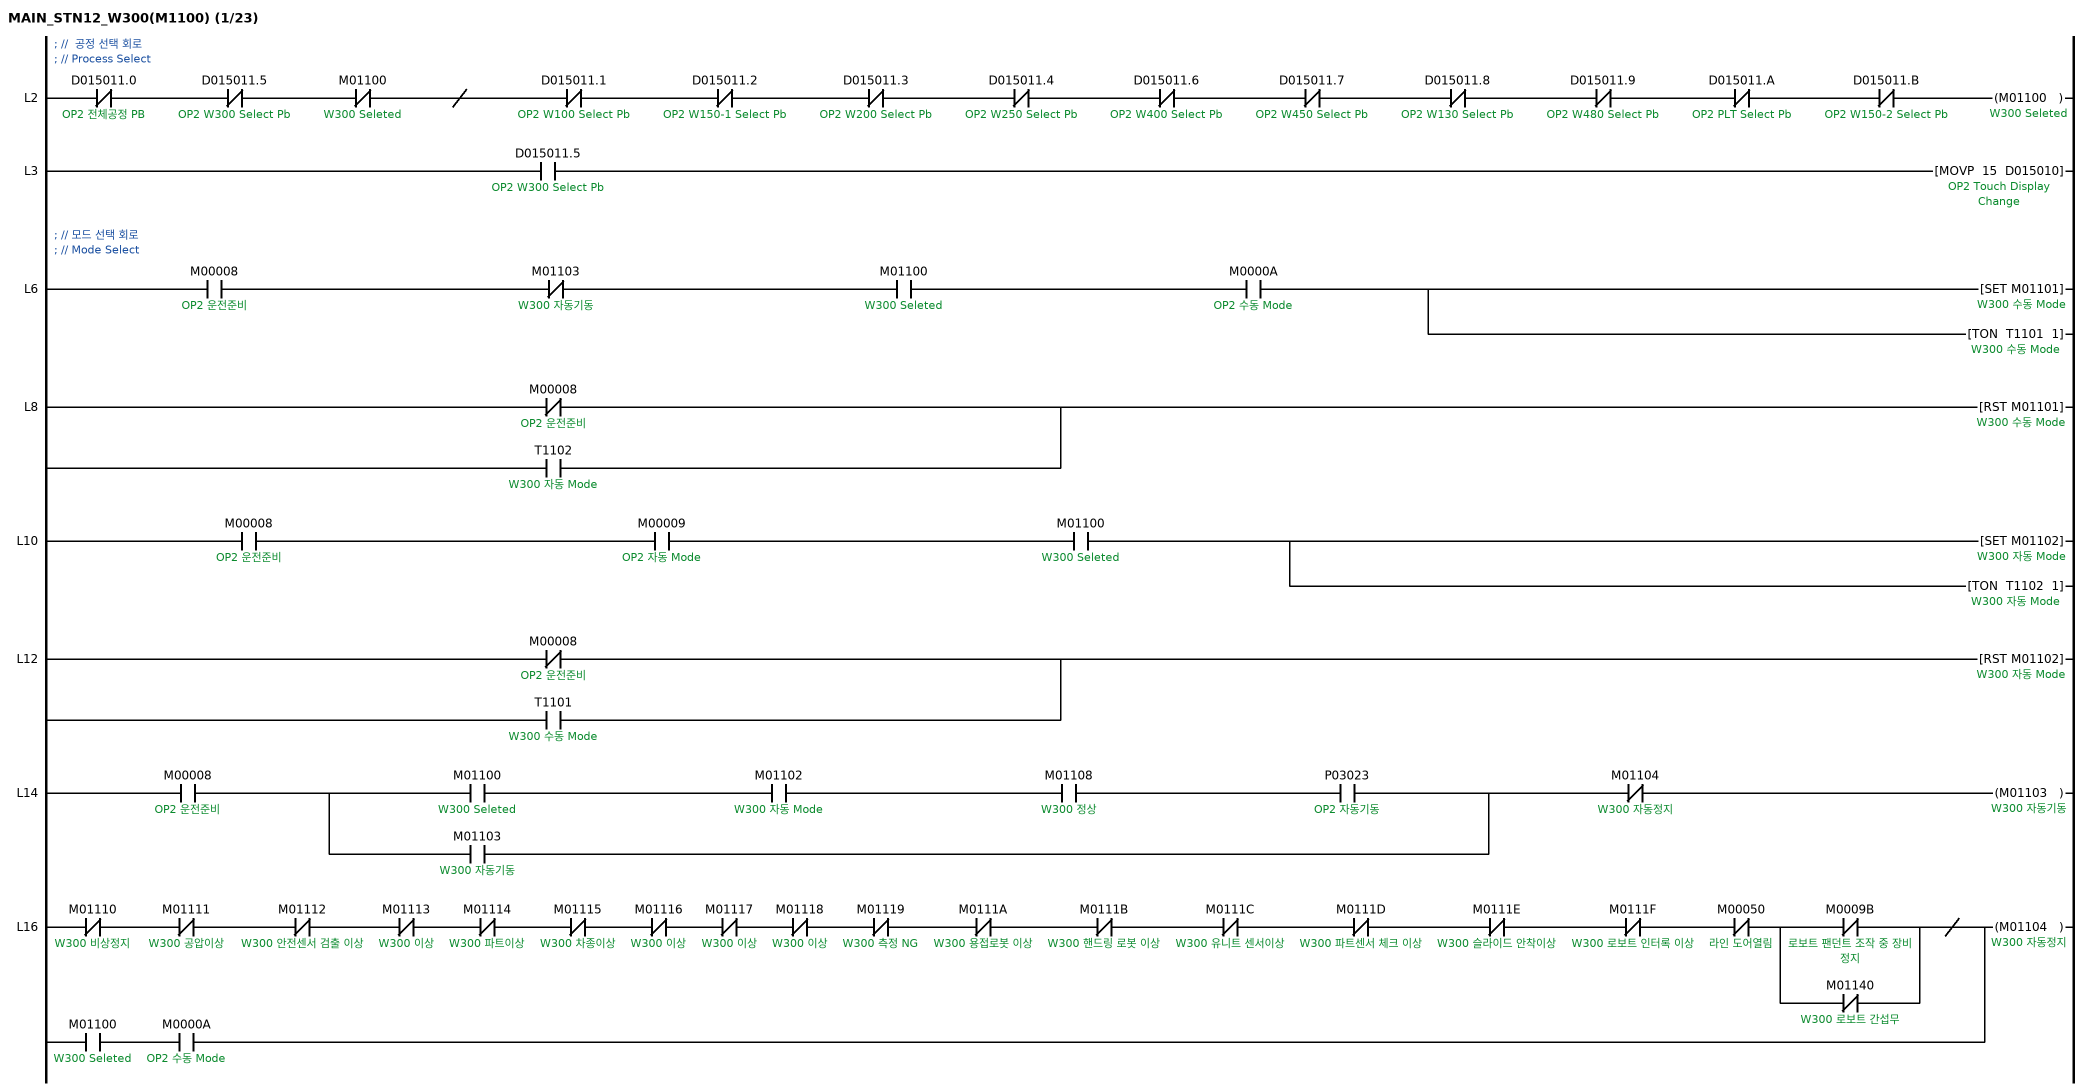
//   //  공정 선택 회로
//   // Process Select
; L2
LOAD NOT  D015011.0	// OP2 전체공정 PB
AND NOT   D015011.5	// OP2 W300 Select Pb
AND NOT   M01100	// W300 Seleted
NOT
AND NOT   D015011.1	// OP2 W100 Select Pb
AND NOT   D015011.2	// OP2 W150-1 Select Pb
AND NOT   D015011.3	// OP2 W200 Select Pb
AND NOT   D015011.4	// OP2 W250 Select Pb
AND NOT   D015011.6	// OP2 W400 Select Pb
AND NOT   D015011.7	// OP2 W450 Select Pb
AND NOT   D015011.8	// OP2 W130 Select Pb
AND NOT   D015011.9	// OP2 W480 Select Pb
AND NOT   D015011.A	// OP2 PLT Select Pb
AND NOT   D015011.B	// OP2 W150-2 Select Pb
OUT       M01100	// W300 Seleted
; L3
LOAD      D015011.5	// OP2 W300 Select Pb
MOVP      15 D015010	// OP2 Touch Display Change
// // 모드 선택 회로
//   // Mode Select
; L6
LOAD      M00008	// OP2 운전준비
AND NOT   M01103	// W300 자동기동
AND       M01100	// W300 Seleted
AND       M0000A	// OP2 수동 Mode
SET       M01101	// W300 수동 Mode
TON       T1101 1	// W300 수동 Mode
; L8
LOAD NOT  M00008	// OP2 운전준비
OR        T1102	// W300 자동 Mode
RST       M01101	// W300 수동 Mode
; L10
LOAD      M00008	// OP2 운전준비
AND       M00009	// OP2 자동 Mode
AND       M01100	// W300 Seleted
SET       M01102	// W300 자동 Mode
TON       T1102 1	// W300 자동 Mode
; L12
LOAD NOT  M00008	// OP2 운전준비
OR        T1101	// W300 수동 Mode
RST       M01102	// W300 자동 Mode
; L14
LOAD      M00008	// OP2 운전준비
LOAD      M01100	// W300 Seleted
AND       M01102	// W300 자동 Mode
AND       M01108	// W300 정상
AND       P03023	// OP2 자동기동
OR        M01103	// W300 자동기동
AND LOAD
AND NOT   M01104	// W300 자동정지
OUT       M01103	// W300 자동기동
; L16
LOAD NOT  M01110	// W300 비상정지
AND NOT   M01111	// W300 공압이상
AND NOT   M01112	// W300 안전센서 검출 이상
AND NOT   M01113	// W300 이상
AND NOT   M01114	// W300 파트이상
AND NOT   M01115	// W300 차종이상
AND NOT   M01116	// W300 이상
AND NOT   M01117	// W300 이상
AND NOT   M01118	// W300 이상
AND NOT   M01119	// W300 측정 NG
AND NOT   M0111A	// W300 용접로봇 이상
AND NOT   M0111B	// W300 핸드링 로봇 이상
AND NOT   M0111C	// W300 유니트 센서이상
AND NOT   M0111D	// W300 파트센서 체크 이상
AND NOT   M0111E	// W300 슬라이드 안착이상
AND NOT   M0111F	// W300 로보트 인터록 이상
AND NOT   M00050	// 라인 도어열림
LOAD NOT  M0009B	// 로보트 팬던트 조작 중 장비 정지
OR NOT    M01140	// W300 로보트 간섭무
AND LOAD
NOT
LOAD      M01100	// W300 Seleted
AND       M0000A	// OP2 수동 Mode
OR LOAD
OUT       M01104	// W300 자동정지

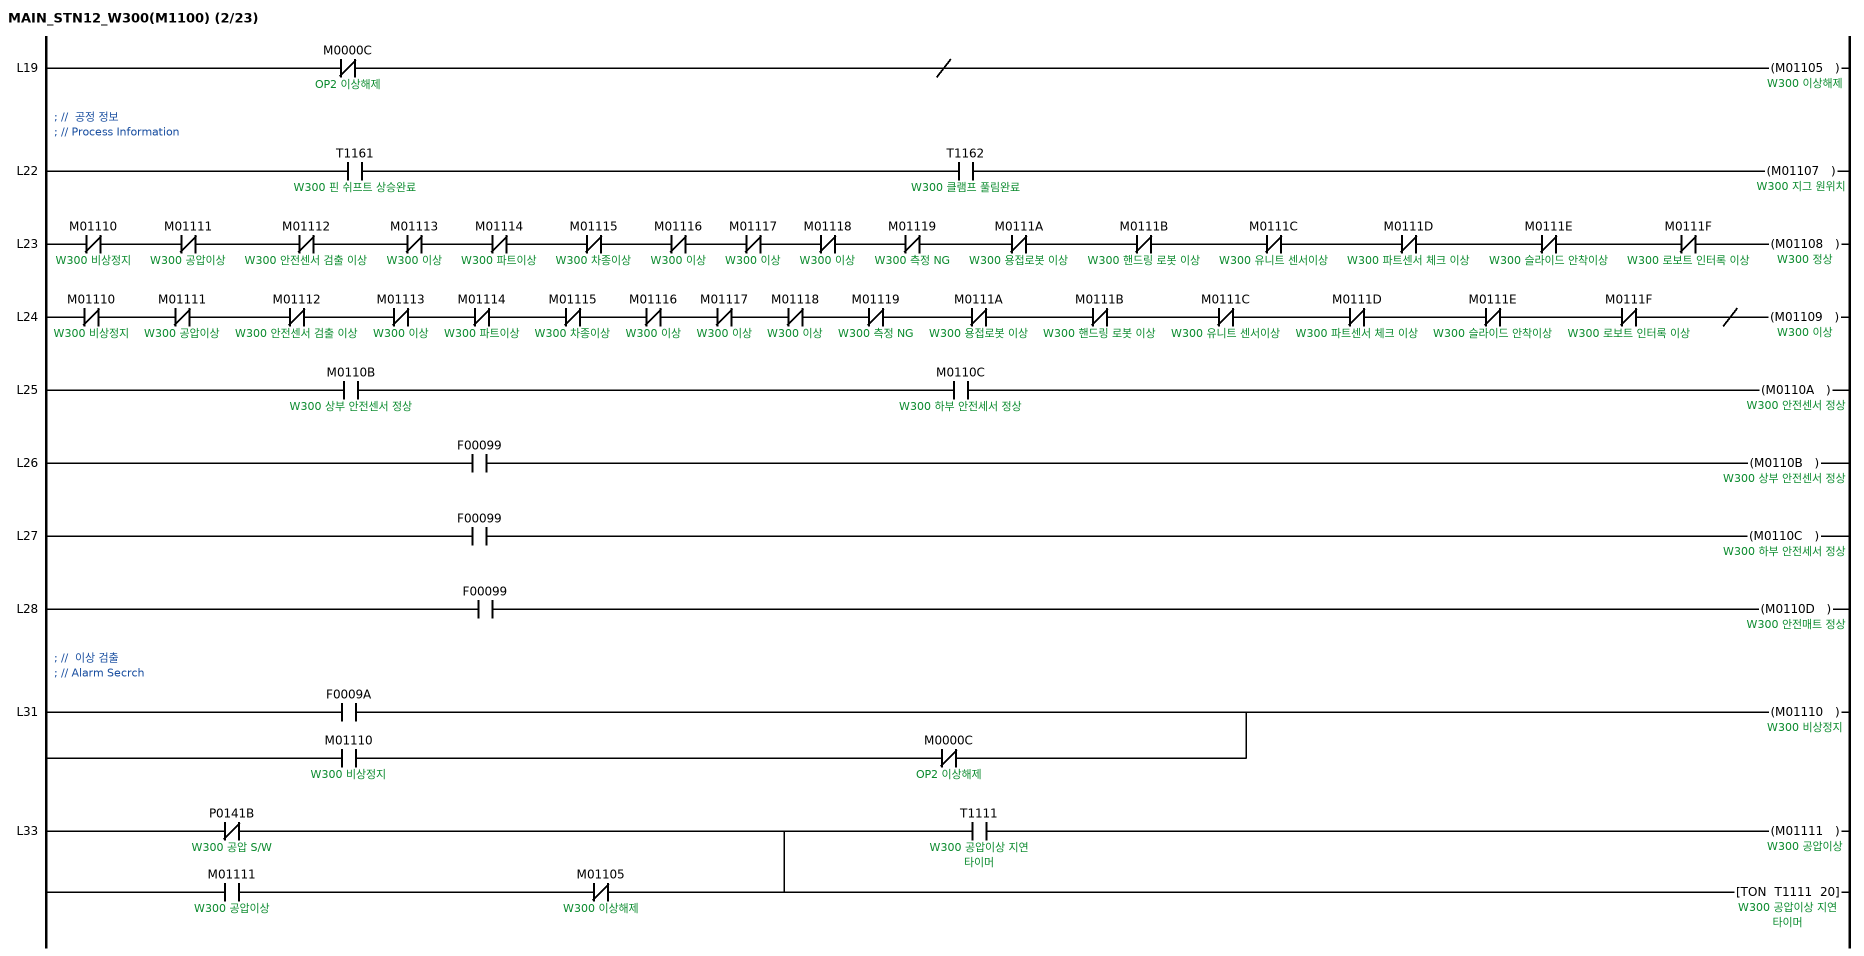
; L19
LOAD NOT  M0000C	// OP2 이상해제
NOT
OUT       M01105	// W300 이상해제
//   //  공정 정보
//   // Process Information
; L22
LOAD      T1161	// W300 핀 쉬프트 상승완료
AND       T1162	// W300 클램프 풀림완료
OUT       M01107	// W300 지그 원위치
; L23
LOAD NOT  M01110	// W300 비상정지
AND NOT   M01111	// W300 공압이상
AND NOT   M01112	// W300 안전센서 검출 이상
AND NOT   M01113	// W300 이상
AND NOT   M01114	// W300 파트이상
AND NOT   M01115	// W300 차종이상
AND NOT   M01116	// W300 이상
AND NOT   M01117	// W300 이상
AND NOT   M01118	// W300 이상
AND NOT   M01119	// W300 측정 NG
AND NOT   M0111A	// W300 용접로봇 이상
AND NOT   M0111B	// W300 핸드링 로봇 이상
AND NOT   M0111C	// W300 유니트 센서이상
AND NOT   M0111D	// W300 파트센서 체크 이상
AND NOT   M0111E	// W300 슬라이드 안착이상
AND NOT   M0111F	// W300 로보트 인터록 이상
OUT       M01108	// W300 정상
; L24
LOAD NOT  M01110	// W300 비상정지
AND NOT   M01111	// W300 공압이상
AND NOT   M01112	// W300 안전센서 검출 이상
AND NOT   M01113	// W300 이상
AND NOT   M01114	// W300 파트이상
AND NOT   M01115	// W300 차종이상
AND NOT   M01116	// W300 이상
AND NOT   M01117	// W300 이상
AND NOT   M01118	// W300 이상
AND NOT   M01119	// W300 측정 NG
AND NOT   M0111A	// W300 용접로봇 이상
AND NOT   M0111B	// W300 핸드링 로봇 이상
AND NOT   M0111C	// W300 유니트 센서이상
AND NOT   M0111D	// W300 파트센서 체크 이상
AND NOT   M0111E	// W300 슬라이드 안착이상
AND NOT   M0111F	// W300 로보트 인터록 이상
NOT
OUT       M01109	// W300 이상
; L25
LOAD      M0110B	// W300 상부 안전센서 정상
AND       M0110C	// W300 하부 안전세서 정상
OUT       M0110A	// W300 안전센서 정상
; L26
LOAD      F00099
OUT       M0110B	// W300 상부 안전센서 정상
; L27
LOAD      F00099
OUT       M0110C	// W300 하부 안전세서 정상
; L28
LOAD      F00099
OUT       M0110D	// W300 안전매트 정상
//   //  이상 검출
//   // Alarm Secrch
; L31
LOAD      F0009A
LOAD      M01110	// W300 비상정지
AND NOT   M0000C	// OP2 이상해제
OR LOAD
OUT       M01110	// W300 비상정지
; L33
LOAD NOT  P0141B	// W300 공압 S/W
LOAD      M01111	// W300 공압이상
AND NOT   M01105	// W300 이상해제
OR LOAD
MPUSH
AND       T1111	// W300 공압이상 지연 타이머
OUT       M01111	// W300 공압이상
MPOP
TON       T1111 20	// W300 공압이상 지연 타이머

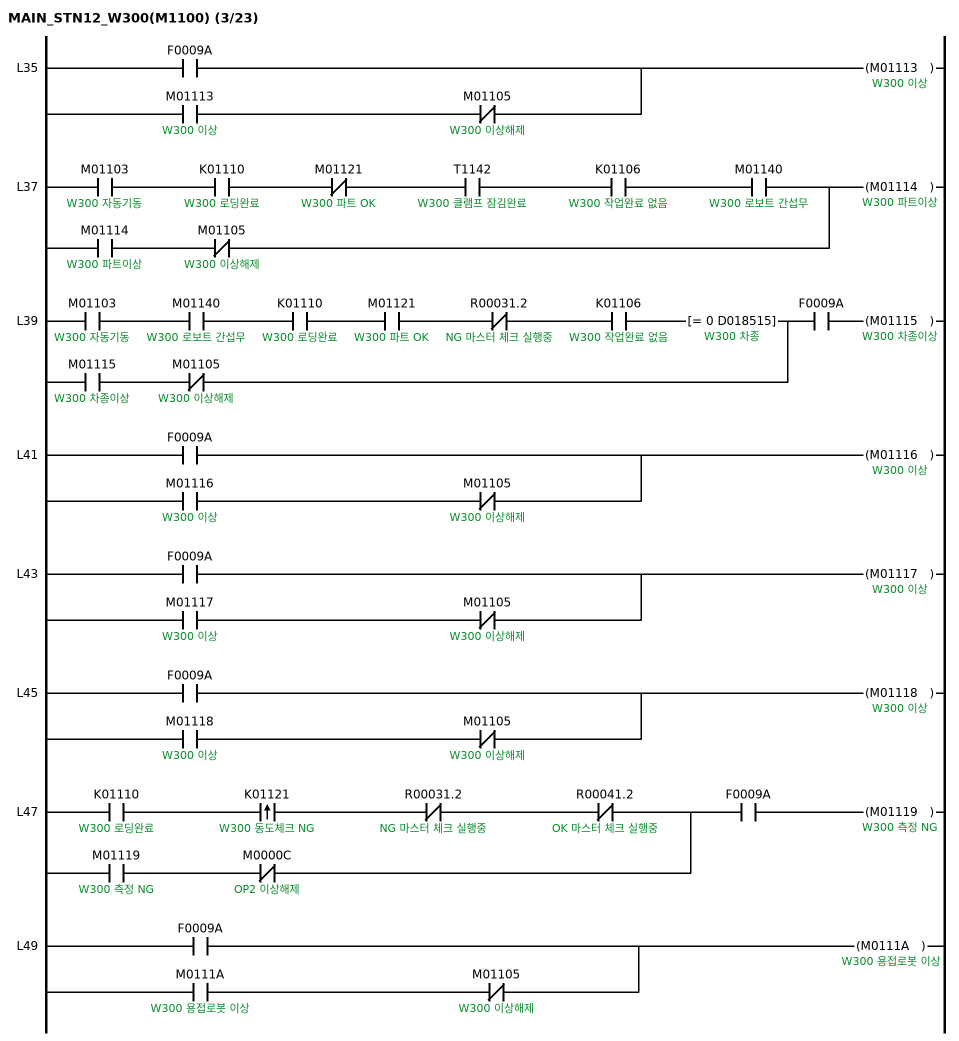
; L35
LOAD      F0009A
LOAD      M01113	// W300 이상
AND NOT   M01105	// W300 이상해제
OR LOAD
OUT       M01113	// W300 이상
; L37
LOAD      M01103	// W300 자동기동
AND       K01110	// W300 로딩완료
AND NOT   M01121	// W300 파트 OK
AND       T1142	// W300 클램프 잠김완료
AND       K01106	// W300 작업완료 없음
AND       M01140	// W300 로보트 간섭무
LOAD      M01114	// W300 파트이상
AND NOT   M01105	// W300 이상해제
OR LOAD
OUT       M01114	// W300 파트이상
; L39
LOAD      M01103	// W300 자동기동
AND       M01140	// W300 로보트 간섭무
AND       K01110	// W300 로딩완료
AND       M01121	// W300 파트 OK
AND NOT   R00031.2	// NG 마스터 체크 실행중
AND       K01106	// W300 작업완료 없음
AND=      0 D018515	// W300 차종
LOAD      M01115	// W300 차종이상
AND NOT   M01105	// W300 이상해제
OR LOAD
AND       F0009A
OUT       M01115	// W300 차종이상
; L41
LOAD      F0009A
LOAD      M01116	// W300 이상
AND NOT   M01105	// W300 이상해제
OR LOAD
OUT       M01116	// W300 이상
; L43
LOAD      F0009A
LOAD      M01117	// W300 이상
AND NOT   M01105	// W300 이상해제
OR LOAD
OUT       M01117	// W300 이상
; L45
LOAD      F0009A
LOAD      M01118	// W300 이상
AND NOT   M01105	// W300 이상해제
OR LOAD
OUT       M01118	// W300 이상
; L47
LOAD      K01110	// W300 로딩완료
ANDP      K01121	// W300 동도체크 NG
AND NOT   R00031.2	// NG 마스터 체크 실행중
AND NOT   R00041.2	// OK 마스터 체크 실행중
LOAD      M01119	// W300 측정 NG
AND NOT   M0000C	// OP2 이상해제
OR LOAD
AND       F0009A
OUT       M01119	// W300 측정 NG
; L49
LOAD      F0009A
LOAD      M0111A	// W300 용접로봇 이상
AND NOT   M01105	// W300 이상해제
OR LOAD
OUT       M0111A	// W300 용접로봇 이상

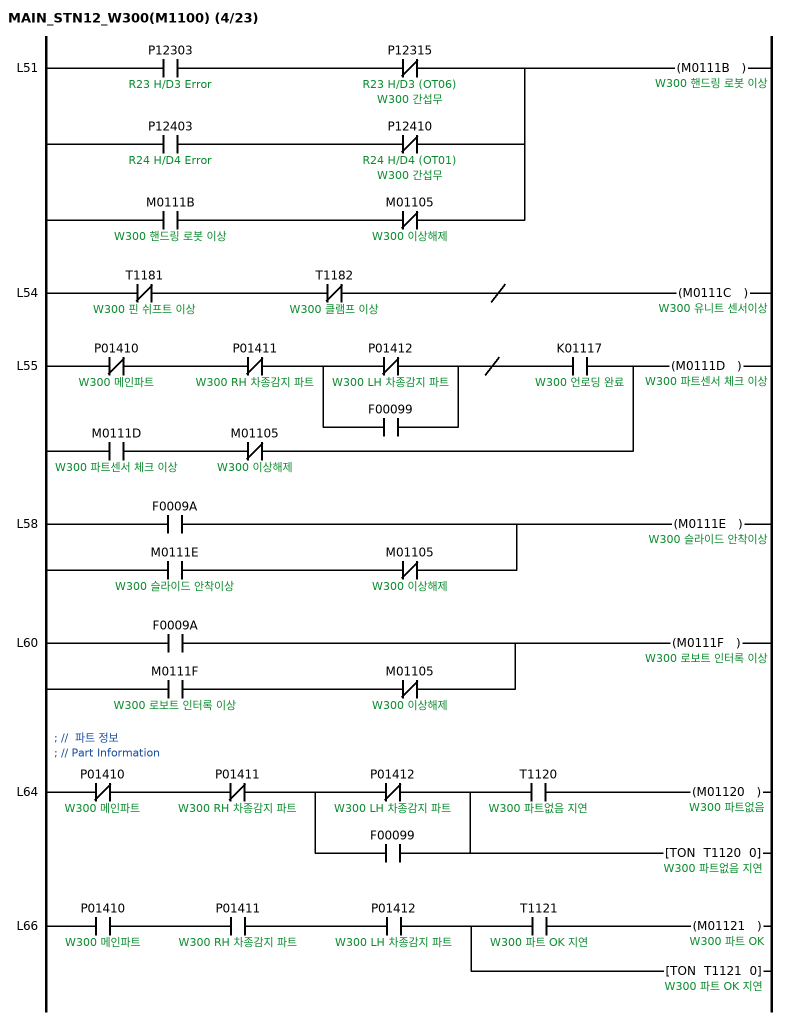
; L51
LOAD      P12303	// R23 H/D3 Error
AND NOT   P12315	// R23 H/D3 (OT06) W300 간섭무
LOAD      P12403	// R24 H/D4 Error
AND NOT   P12410	// R24 H/D4 (OT01) W300 간섭무
OR LOAD
LOAD      M0111B	// W300 핸드링 로봇 이상
AND NOT   M01105	// W300 이상해제
OR LOAD
OUT       M0111B	// W300 핸드링 로봇 이상
; L54
LOAD NOT  T1181	// W300 핀 쉬프트 이상
AND NOT   T1182	// W300 클램프 이상
NOT
OUT       M0111C	// W300 유니트 센서이상
; L55
LOAD NOT  P01410	// W300 메인파트
AND NOT   P01411	// W300 RH 차종감지 파트
LOAD NOT  P01412	// W300 LH 차종감지 파트
OR        F00099
AND LOAD
NOT
AND       K01117	// W300 언로딩 완료
LOAD      M0111D	// W300 파트센서 체크 이상
AND NOT   M01105	// W300 이상해제
OR LOAD
OUT       M0111D	// W300 파트센서 체크 이상
; L58
LOAD      F0009A
LOAD      M0111E	// W300 슬라이드 안착이상
AND NOT   M01105	// W300 이상해제
OR LOAD
OUT       M0111E	// W300 슬라이드 안착이상
; L60
LOAD      F0009A
LOAD      M0111F	// W300 로보트 인터록 이상
AND NOT   M01105	// W300 이상해제
OR LOAD
OUT       M0111F	// W300 로보트 인터록 이상
//   //  파트 정보
//   // Part Information
; L64
LOAD NOT  P01410	// W300 메인파트
AND NOT   P01411	// W300 RH 차종감지 파트
LOAD NOT  P01412	// W300 LH 차종감지 파트
OR        F00099
AND LOAD
MPUSH
AND       T1120	// W300 파트없음 지연
OUT       M01120	// W300 파트없음
MPOP
TON       T1120 0	// W300 파트없음 지연
; L66
LOAD      P01410	// W300 메인파트
AND       P01411	// W300 RH 차종감지 파트
AND       P01412	// W300 LH 차종감지 파트
MPUSH
AND       T1121	// W300 파트 OK 지연
OUT       M01121	// W300 파트 OK
MPOP
TON       T1121 0	// W300 파트 OK 지연

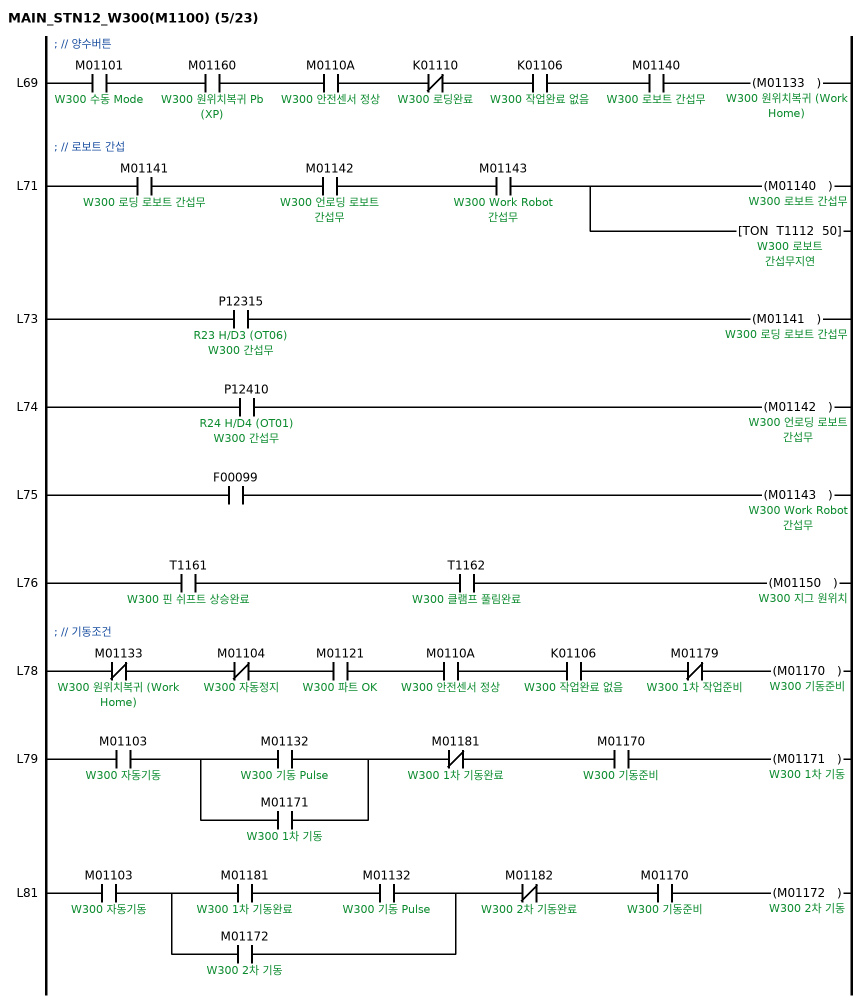
//   // 양수버튼
; L69
LOAD      M01101	// W300 수동 Mode
AND       M01160	// W300 원위치복귀 Pb (XP)
AND       M0110A	// W300 안전센서 정상
AND NOT   K01110	// W300 로딩완료
AND       K01106	// W300 작업완료 없음
AND       M01140	// W300 로보트 간섭무
OUT       M01133	// W300 원위치복귀 (Work Home)
//   // 로보트 간섭
; L71
LOAD      M01141	// W300 로딩 로보트 간섭무
AND       M01142	// W300 언로딩 로보트 간섭무
AND       M01143	// W300 Work Robot 간섭무
OUT       M01140	// W300 로보트 간섭무
TON       T1112 50	// W300 로보트 간섭무지연
; L73
LOAD      P12315	// R23 H/D3 (OT06) W300 간섭무
OUT       M01141	// W300 로딩 로보트 간섭무
; L74
LOAD      P12410	// R24 H/D4 (OT01) W300 간섭무
OUT       M01142	// W300 언로딩 로보트 간섭무
; L75
LOAD      F00099
OUT       M01143	// W300 Work Robot 간섭무
; L76
LOAD      T1161	// W300 핀 쉬프트 상승완료
AND       T1162	// W300 클램프 풀림완료
OUT       M01150	// W300 지그 원위치
//   // 기동조건
; L78
LOAD NOT  M01133	// W300 원위치복귀 (Work Home)
AND NOT   M01104	// W300 자동정지
AND       M01121	// W300 파트 OK
AND       M0110A	// W300 안전센서 정상
AND       K01106	// W300 작업완료 없음
AND NOT   M01179	// W300 1차 작업준비
OUT       M01170	// W300 기동준비
; L79
LOAD      M01103	// W300 자동기동
LOAD      M01132	// W300 기동 Pulse
OR        M01171	// W300 1차 기동
AND LOAD
AND NOT   M01181	// W300 1차 기동완료
AND       M01170	// W300 기동준비
OUT       M01171	// W300 1차 기동
; L81
LOAD      M01103	// W300 자동기동
LOAD      M01181	// W300 1차 기동완료
AND       M01132	// W300 기동 Pulse
OR        M01172	// W300 2차 기동
AND LOAD
AND NOT   M01182	// W300 2차 기동완료
AND       M01170	// W300 기동준비
OUT       M01172	// W300 2차 기동

